// TwinCAT 3 PLC project SPS_1
// ProgramVersion: 3.1.4026.10
// CompilerDefines: VISU_USEPROPERTYINFO
// libraries:
//   Tc2_ModbusRTU, * (Beckhoff Automation GmbH)
//   Tc2_Standard, * (Beckhoff Automation GmbH)
//   Tc2_System, * (Beckhoff Automation GmbH)
//   Tc2_TcpIp, * (Beckhoff Automation GmbH)
//   Tc2_Utilities, * (Beckhoff Automation GmbH)
// project tree:
//   DUTs/01_Liste/01_Zustände/ eObjectAktorState.TcDUT, eSequenceState.TcDUT, eSkillState.TcDUT, eSystemState.TcDUT
//   DUTs/01_Liste/02_Commands/ eSkillCommand.TcDUT, eSystemCommand.TcDUT
//   DUTs/01_Liste/03_Konfiguration/ eRobMoveType.TcDUT, eRobPosType.TcDUT
//   DUTs/02_Schnittstellen/ I_State_Skill.TcIO, I_State_Object.TcIO
//   DUTs/03_Strukturen/01_Schnittstellen/ sKraftVariablen.TcDUT, sRoboterProzessVariablen.TcDUT, sSmartGreiferProzessVariablen.TcDUT
//   DUTs/03_Strukturen/02_Objektintern/01_FB_Roboter/ sPositionArrays.TcDUT, sPositionValues.TcDUT, sRealTimeData.TcDUT
//   DUTs/03_Strukturen/02_Objektintern/02_FB_Kraftsensor/ Kraftvariablen.TcDUT (not stored), Request.TcDUT, Response_Parameters.TcDUT, Response_Values.TcDUT
//   DUTs/04_Union/ Array2_Int.TcDUT, Array8_LReal.TcDUT, Int_2Byte.TcDUT, String_Array256.TcDUT
//   / GlobalTextList.TcGTLO, PlcTask.TcTTO, Visualization Manager.TcVMO (not stored), VISU_TASK.TcTTO
//   GVLs/ GVL.TcGVL
//   POUs/01_Prozessmodell/01_Skills/01_Grundstruktur/ GrundstrukturSkill.TcPOU
//   POUs/01_Prozessmodell/01_Skills/02_Skills/00_Referenz/ Basis_Skill.TcPOU
//   POUs/01_Prozessmodell/01_Skills/02_Skills/01_Roboter/ Skill_Position_anfahren.TcPOU (not stored), Skill_Position_anfahren_erweitert.TcPOU
//   POUs/01_Prozessmodell/01_Skills/02_Skills/02_Greifer/ Skill_Greifer_Oeffnen.TcPOU, Skill_Greifer_Pos_Anfahren.TcPOU, Skill_Greifer_Schliessen.TcPOU
//   POUs/01_Prozessmodell/02_Sequenzen/ Seq_1.TcPOU, Seq_2.TcPOU
//   POUs/02_Anlagenmodell/01_Grundstruktur/ GrundstrukturObjekt.TcPOU
//   POUs/02_Anlagenmodell/02_Objektklassen/00_Referenz/ Basis_Objekt.TcPOU
//   POUs/02_Anlagenmodell/02_Objektklassen/ FB_Kraftsensor.TcPOU, FB_Roboter.TcPOU, FB_SmartGreifer.TcPOU
//   POUs/02_Anlagenmodell/ Anlage.TcPOU
//   POUs/03_Systemmodell/ Systemparameter.TcPOU, Zustandshandling.TcPOU
//   POUs/ MAIN.TcPOU
//   VISUs/00_Debug/ SystemState.TcVIS
// real-time tasks:
//   TASK PlcTask: cycle T#10ms, priority 20, ADS port 350
//   TASK VISU_TASK: cycle T#200000us, priority 30, ADS port 351
//   TASK PlcTask1: cycle T#10ms, priority 21, ADS port 352
//   TASK PlcTask2: cycle T#10ms, priority 22, ADS port 353
// I/O:
//   DEVICE Gerät 1 (EtherCAT), AmsNetId 147.87.172.51.2.1
//     Box 1 (BK1120)
// variable links:
//   SPS_3/SPS_3 Instance <-> Device 1 (EtherCAT)/Box 1 (BK1120)
//     PlcTask Inputs/Anlage.Gripper.Communication.InData/D[{0..21}] <-> Term 2 (KL6041)/Channel 1/Data In {0..21}  (22 links)
//     PlcTask Inputs/Anlage.Gripper.Communication.InData/Status <-> Term 2 (KL6041)/Channel 1/Status
//     PlcTask Outputs/Anlage.Gripper.Communication.OutData/Ctrl <-> Term 2 (KL6041)/Channel 1/Ctrl
//     PlcTask Outputs/Anlage.Gripper.Communication.OutData/D[{0..21}] <-> Term 2 (KL6041)/Channel 1/Data Out {0..21}  (22 links)

CONFIGURATION SPS_1
    RESOURCE PLC ON TwinCAT3
        TASK PlcTask(INTERVAL := T#10ms, PRIORITY := 20);
        TASK VISU_TASK(INTERVAL := T#200000us, PRIORITY := 30);
        PROGRAM MAIN WITH PlcTask : MAIN;
        PROGRAM VisuElems_Visu_Prg WITH VISU_TASK : VisuElems.Visu_Prg;
    END_RESOURCE
END_CONFIGURATION

// ---- DUTs/01_Liste/01_Zustände/eObjectAktorState.TcDUT
{attribute 'qualified_only'}
{attribute 'strict'}
{attribute 'to_string'}
TYPE eObjectAktorState :
(
	AUS 					:= 0,				// Das Objekt ist ausgeschalten
	BEREIT 					:= 1,				// Das Objekt ist eingeschalten und bereit
	MANUELL					:= 2,				// Das Objekt befindet sich im Manuell-Modus
	LAUFEND 				:= 3,				// Das Objekt ist aktiv
	ABGESCHLOSSEN_INTERN 	:= 4,				// Das Objekt hat den Prozess durchgeführt und hat selbständig gestoppt
	ABGESCHLOSSEN_EXTERN	:= 5,				// Das Objekt wurde durch den Skill gestoppt (ERREICHT / LIMIT)
	GESTOPPT 				:= 6,				// Das Objekt wurde durch das System gestoppt
	FEHLER					:= 7				// Es gibt einen Fehler bezüglich des Objektes
);
END_TYPE

// ---- DUTs/01_Liste/01_Zustände/eSequenceState.TcDUT
{attribute 'qualified_only'}
{attribute 'strict'}
{attribute 'to_string'}
TYPE eSequenceState  :
(
	BEREIT	 		:= 0,				// Der Skill ist bereit einen Prozess auszuführen (Startzustand)
	LAUFEND 		:= 1,				// Der Skill führt einen Prozess aus
	ABGESCHLOSSEN 	:= 2,				// Der Prozess wurde abgeschlossen (Durch Objekt abgeschlossen)
	FEHLER			:= 3				// Es gibt einen Fehler bezüglich des Prozesses 
);
END_TYPE

// ---- DUTs/01_Liste/01_Zustände/eSkillState.TcDUT
{attribute 'qualified_only'}
{attribute 'strict'}
{attribute 'to_string'}
TYPE eSkillState :
(
	BEREIT	 		:= 0,				// Der Skill ist bereit einen Prozess auszuführen (Startzustand)
	LAUFEND 		:= 1,				// Der Skill führt einen Prozess aus
	ABGESCHLOSSEN 	:= 2,				// Der Prozess wurde abgeschlossen (Durch Objekt abgeschlossen)
	FEHLER			:= 3,				// Es gibt einen Fehler bezüglich des Prozesses 
	LIMITE			:= 4,				// Grenzwert wurde überschritten und Prozess wurde abgebrochen
	ERREICHT		:= 5				// Prozessziel wurde erreicht und Prozess wurde durch Skill beendet  
);	
END_TYPE

// ---- DUTs/01_Liste/01_Zustände/eSystemState.TcDUT
{attribute 'qualified_only'}
{attribute 'strict'}
{attribute 'to_string'}
TYPE eSystemState :
(
	AUS 			:= 0,				// Das System ist ausgeschalten
	BEREIT 			:= 1,				// Das System ist eingeschalten und bereit einen Prozess durchzuführen
	LAUFEND 		:= 2,				// Ein Prozess wird ausgeführt
	GESTOPPT		:= 3,				// Ein Prozess wurde gestoppt
	FEHLER			:= 4				// Es gibt einen Fehler im System 
);
END_TYPE

// ---- DUTs/01_Liste/02_Commands/eSkillCommand.TcDUT
{attribute 'qualified_only'}
{attribute 'strict'}
{attribute 'to_string'}
TYPE eSkillCommand :
(
	KEINE		:= 0,
	STARTEN		:= 1,
	STOPPEN		:= 2,
	RESETTEN 	:= 3
);
END_TYPE

// ---- DUTs/01_Liste/02_Commands/eSystemCommand.TcDUT
{attribute 'qualified_only'}
{attribute 'strict'}
{attribute 'to_string'}
TYPE eSystemCommand :
(
	KEINE		:= 0,
	AUSCHALTEN 	:= 1,
	EINSCHALTEN := 2,
	STOPPEN		:= 3,
	RESETTEN	:= 4
);
END_TYPE

// ---- DUTs/01_Liste/03_Konfiguration/eRobMoveType.TcDUT
{attribute 'qualified_only'}
{attribute 'strict'}
{attribute 'to_string'}
TYPE eRobMoveType :
(
	LinearToolSpace 			:= 0,		// Move to position (linear in tool-space)
	LinearJointSpace 			:= 1,		// Move to position (linear in joint-space)
	CircularToolSpace 			:= 2,		// Move Circular: Move to position (circular in tool-space)
	BlendCircularMoveLinear		:= 3		// Move Process
);
END_TYPE

// ---- DUTs/01_Liste/03_Konfiguration/eRobPosType.TcDUT
{attribute 'qualified_only'}
{attribute 'strict'}
{attribute 'to_string'}
TYPE eRobPosType :
(
	Absolut := 0,			// Absolute Bewegung bezogen auf Basis-Koordinatensystem
	Relativ := 1			// Relative Bewegung bezogen auf aktuelle Position
);
END_TYPE

// ---- DUTs/03_Strukturen/01_Schnittstellen/sKraftVariablen.TcDUT
TYPE sKraftVariablen :
STRUCT
	Fx					:LREAL;							// Kraft in X-Richtung 
	Fy					:LREAL;							// Kraft in Y-Richtung 
	Fz					:LREAL;							// Kraft in Z-Richtung 
END_STRUCT
END_TYPE

// ---- DUTs/03_Strukturen/01_Schnittstellen/sRoboterProzessVariablen.TcDUT
TYPE sRoboterProzessVariablen :
STRUCT
	q1					:LREAL;				// X-Koordinate oder Gelenkwinkel 1
	q2					:LREAL;				// Y-Koordinate oder Gelenkwinkel 2
	q3					:LREAL;				// Z-Koordinate oder Gelenkwinkel 3
	q4					:LREAL;				// Orintierung um X-Achse oder Gelenkwinkel 4
	q5					:LREAL;				// Orientierung um Y-Achse oder Gelenkwinkel 5
	q6					:LREAL;				// Orientierung um Z-Achse oder Gelenkwinkel 6
	v					:LREAL;				// Geschwindigkeit
	a					:LREAL;				// Beschleunigung
	PosTyp				:eRobPosType;		// Position-Typ definieren (Absolut / Relativ)		
	MoveTyp				:eRobMoveType;		// Bewegungsart definieren (Linear / Circular etc.)
END_STRUCT
END_TYPE

// ---- DUTs/03_Strukturen/01_Schnittstellen/sSmartGreiferProzessVariablen.TcDUT
TYPE sSmartGreiferProzessVariablen :
STRUCT
	Pos				:USINT;			// Position von Greifer in mm
	Geschw			:USINT;			// Geschwindigkeit in %
	F				:USINT;			// Kraft in %
END_STRUCT
	
END_TYPE

// ---- DUTs/03_Strukturen/02_Objektintern/01_FB_Roboter/sPositionArrays.TcDUT
TYPE sPositionArrays :
STRUCT
	q1		: ARRAY[0..7] OF BYTE;
	q2		: ARRAY[0..7] OF BYTE;
	q3		: ARRAY[0..7] OF BYTE;
	q4		: ARRAY[0..7] OF BYTE;
	q5		: ARRAY[0..7] OF BYTE;
	q6		: ARRAY[0..7] OF BYTE;
END_STRUCT
END_TYPE

// ---- DUTs/03_Strukturen/02_Objektintern/01_FB_Roboter/sPositionValues.TcDUT
TYPE sPositionValues :
STRUCT
	q1			:LREAL;
	q2			:LREAL;
	q3			:LREAL;
	q4			:LREAL;
	q5			:LREAL;
	q6			:LREAL;
END_STRUCT
END_TYPE

// ---- DUTs/03_Strukturen/02_Objektintern/01_FB_Roboter/sRealTimeData.TcDUT
TYPE sRealTimeData :
STRUCT
	messageSize 				: ARRAY[0..3] OF BYTE;
	
	timestamp 					: ARRAY[0..7] OF BYTE;
	
	//qTarget 					: ARRAY[0..47] OF BYTE;
	qTargetQ1 					: ARRAY[0..7] OF BYTE;
	qTargetQ2 					: ARRAY[0..7] OF BYTE;
	qTargetQ3 					: ARRAY[0..7] OF BYTE;
	qTargetQ4 					: ARRAY[0..7] OF BYTE;
	qTargetQ5 					: ARRAY[0..7] OF BYTE;
	qTargetQ6 					: ARRAY[0..7] OF BYTE;
	
	qdTarget 					: ARRAY[0..47] OF BYTE;
	
	qddTarget 					: ARRAY[0..47] OF BYTE;
	
	iTarget 					: ARRAY[0..47] OF BYTE;
	
	mTarget 					: ARRAY[0..47] OF BYTE;
	
	//qActual 					: ARRAY[0..47] OF BYTE;
	qActualQ1 					: ARRAY[0..7] OF BYTE;
	qActualQ2 					: ARRAY[0..7] OF BYTE;
	qActualQ3 					: ARRAY[0..7] OF BYTE;
	qActualQ4 					: ARRAY[0..7] OF BYTE;
	qActualQ5 					: ARRAY[0..7] OF BYTE;
	qActualQ6 					: ARRAY[0..7] OF BYTE;
	
	//qdActual 					: ARRAY[0..47] OF BYTE;
	qdActualQ1 					: ARRAY[0..7] OF BYTE;
	qdActualQ2 					: ARRAY[0..7] OF BYTE;
	qdActualQ3 					: ARRAY[0..7] OF BYTE;
	qdActualQ4 					: ARRAY[0..7] OF BYTE;
	qdActualQ5 					: ARRAY[0..7] OF BYTE;
	qdActualQ6 					: ARRAY[0..7] OF BYTE;
	
	iActual 					: ARRAY[0..47] OF BYTE;
	
	toolAccelerometerValues 	: ARRAY[0..23] OF BYTE;
	
	unused_1					: ARRAY[0..119] OF BYTE;
	
	tcpForce 					: ARRAY[0..47] OF BYTE;
	
	//toolVector 					: ARRAY[0..47] OF BYTE;
	toolVectorQ1 				: ARRAY[0..7] OF BYTE;
	toolVectorQ2 				: ARRAY[0..7] OF BYTE;
	toolVectorQ3 				: ARRAY[0..7] OF BYTE;
	toolVectorQ4 				: ARRAY[0..7] OF BYTE;
	toolVectorQ5 				: ARRAY[0..7] OF BYTE;
	toolVectorQ6 				: ARRAY[0..7] OF BYTE;
	
	tcpSpeed 					: ARRAY[0..47] OF BYTE;
	
	digitalInputBits 			: ARRAY[0..7] OF BYTE;
	
	unused_2					: ARRAY[0..119] OF BYTE;
END_STRUCT
END_TYPE

// ---- DUTs/03_Strukturen/02_Objektintern/02_FB_Kraftsensor/Request.TcDUT
TYPE Request :
STRUCT
	Command			:UINT;		// Value according to the command table
	Data			:ARRAY[0..18] OF UINT := [0];		
END_STRUCT
END_TYPE

// ---- DUTs/03_Strukturen/02_Objektintern/02_FB_Kraftsensor/Response_Parameters.TcDUT
TYPE Response_Parameters :
STRUCT
	Header				:UINT;			// Fixed 0x1234
	Unit_Force			:USINT;			// The unit of the calculated Force values
	Unit_Torque			:USINT;			// The unit of the calculated Torque values
	CPF					:UDINT;			// Counts per Force value
	CPT					:UDINT;			// Counts per Torque value
	ScaleFactorFx		:UINT;			// Additional scaling factor (for the Fx,Fy,Fz,Tx,Ty,Tz)
	ScaleFactorFy		:UINT;			// Additional scaling factor (for the Fx,Fy,Fz,Tx,Ty,Tz)
	ScaleFactorFz		:UINT;			// Additional scaling factor (for the Fx,Fy,Fz,Tx,Ty,Tz)
	ScaleFactorTx		:UINT;			// Additional scaling factor (for the Fx,Fy,Fz,Tx,Ty,Tz)
	ScaleFactorTy		:UINT;			// Additional scaling factor (for the Fx,Fy,Fz,Tx,Ty,Tz)
	ScaleFactorTz		:UINT;			// Additional scaling factor (for the Fx,Fy,Fz,Tx,Ty,Tz)
END_STRUCT
END_TYPE

// ---- DUTs/03_Strukturen/02_Objektintern/02_FB_Kraftsensor/Response_Values.TcDUT
TYPE Response_Values :
STRUCT
	Header				:UINT;			// Fixed 0x1234
	Status				:UINT;			// Status word of the sensor and Compute Box
	Fx					:INT;			// X-axis force in 32 bit Counts*
	Fy					:INT;			// Y-axis force in 32 bit Counts*
	Fz					:INT;			// Z-axis force in 32 bit Counts*
	Tx					:INT;			// X-axis torque in 32 bit Counts* (0 if not available)
	Ty					:INT;			// Y-axis torque in 32 bit Counts* (0 if not available)
	Tz					:INT;			// Z-axis torque in 32 bit Counts* (0 if not available)
END_STRUCT
END_TYPE

// ---- DUTs/04_Union/Array2_Int.TcDUT
TYPE Array2_Int :
UNION
	arrByte 		:ARRAY[0..1] OF BYTE;
	sValue			:INT; 
END_UNION
END_TYPE

// ---- DUTs/04_Union/Array8_LReal.TcDUT
TYPE Array8_LReal :
UNION
	arrByte			:ARRAY[0..7] OF BYTE;
	rValue			:LREAL;
END_UNION
END_TYPE

// ---- DUTs/04_Union/Int_2Byte.TcDUT
TYPE Int_2Byte :
UNION
	sValue			:INT; 
	arrByte 		:ARRAY[0..1] OF BYTE;
END_UNION
END_TYPE

// ---- DUTs/04_Union/String_Array256.TcDUT
TYPE String_Array256 :
UNION
	sValue			:STRING; 
	arrByte 		:ARRAY[0..255] OF BYTE;
END_UNION
END_TYPE

// ---- GVLs/GVL.TcGVL
{attribute 'qualified_only'}
VAR_GLOBAL
	// Schnittstellenvariablen 
		// System: 
		SystemState								:eSystemState; 
		SystemCommand							:eSystemCommand; 
		Error									:BOOL;
		
		// Kontrollvariablen: 
		Reset									:BOOL;
		
		// Prozessvariablen
		eKraftLimitValue						:sKraftVariablen;
		eKraftErreichtValue						:sKraftVariablen;
		
		
		// SkillStates
		
		// ObjectStates
		Robot_State								:eObjectAktorState;
		Greifer_State							:eObjectAktorState;
		Sensor_State							:eObjectAktorState;
		
			
		
		
		
END_VAR

// ---- DUTs/02_Schnittstellen/I_State_Skill.TcIO
INTERFACE I_State_Skill

PROPERTY P_State : eSkillState
GET
END_GET
END_PROPERTY

END_INTERFACE

// ---- DUTs/02_Schnittstellen/I_State_Object.TcIO
INTERFACE I_State_Object

PROPERTY P_State : eObjectAktorState
GET
END_GET
END_PROPERTY

END_INTERFACE

// ---- POUs/MAIN.TcPOU
PROGRAM MAIN
VAR
	TestAblauf				:Seq_2;
	
	Execute					:BOOL;		
	Position_1				:sRoboterProzessVariablen;
	Position_2				:sRoboterProzessVariablen;
	Position_3				:sRoboterProzessVariablen;

	
	TestSystem				:eSystemCommand; 
	TestSkill				:eSkillCommand; 
	TestVariablen			:sSmartGreiferProzessVariablen;
	
	Param1					:sSmartGreiferProzessVariablen;
	Param2					:sSmartGreiferProzessVariablen;
	Param3					:sSmartGreiferProzessVariablen;
	Param4					:sSmartGreiferProzessVariablen;
		
END_VAR

Zustandshandling();
Anlage();
Systemparameter();


Position_1.q1 := -0.3;
Position_1.q2 := 0.5;
Position_1.q3 := 0.42;
Position_1.q4 := 120;
Position_1.q5 := -132;
Position_1.q6 := 0;
Position_1.a := 0.05;
Position_1.v := 0.05;
Position_1.MoveTyp := 3;
Position_1.PosTyp := 0;

Position_2.q1 := 0.4;
Position_2.q2 := 0.52;
Position_2.q3 := 0.42;
Position_2.q4 := 120;
Position_2.q5 := -132;
Position_2.q6 := 0;
Position_2.a := 0.05;
Position_2.v := 0.05;
Position_2.MoveTyp := 3;
Position_2.PosTyp := 0;

Position_3.q1 := 0.05;
Position_3.q2 := 0.68;
Position_3.q3 := 0.42;
Position_3.q4 := 120;
Position_3.q5 := -132;
Position_3.q6 := 0;
Position_3.a := 0.05;
Position_3.v := 0.05;
Position_3.MoveTyp := 3;
Position_3.PosTyp := 0;

GVL.eKraftLimitValue.Fz := -40;

TestAblauf(
	bExecute := Execute,
	iSysCommand := GVL.SystemCommand,
	Position_1 := Position_1,
	Position_2 := Position_2,
	Position_3 := Position_3);

END_PROGRAM

// ---- POUs/01_Prozessmodell/02_Sequenzen/Seq_2.TcPOU
FUNCTION_BLOCK Seq_2
VAR_INPUT
	// Basis-Inputs
	bExecute			:BOOL;				// Trigger für Ausführung von Sequenz
	iSysCommand			:eSystemCommand;	// Steuerungsvariabel von System (Resetten)
	
	// Prozess-Inputs 
	Position_1			:sRoboterProzessVariablen;
	Position_2			:sRoboterProzessVariablen;
	Position_3			:sRoboterProzessVariablen;
	
END_VAR
VAR_OUTPUT
	bDone				:BOOL;				// Information ob Sequenz ausgfeührt wurde
	bBusy				:BOOL;				// Information ob Sequenz im Moment ausgeführt wird
	bError				:BOOL;				// Information ob sich Sequenz in Fehlerzustand befindet
END_VAR
VAR
	// Sequenz-Zustände
	iState				:eSequenceState;
	
	// Startvariablen (FB soll nur bei einer steigenden Flanke gestartet werden)
	fTrigger			:R_TRIG;			// Erkennung einer steigenden Flanke für den Starte
	fSwitch				:SR;				// Setzen des Signals
	bSwitchResett		:BOOL;				// Resetten des Signals
	
	// Zustandsvariablen
	bStarten			:BOOL;
	bStoppen			:BOOL;
	bResetten			:BOOL;
	
	// Management-Variablen:
	bFinished			:BOOL;
	bInit				:BOOL;
	
	// Skill-Instanziierungen
	P2P_Movement		:Skill_Position_anfahren_erweitert;
	Position			:sRoboterProzessVariablen;
END_VAR

// Aufrufen von Skills und Ablauf
Ablauf();	
Skills();

//_______________________________________________________________
// Reaktion auf Fehler
IF bError THEN
	iState := 3;
END_IF	

// Reaktion auf Input-Variablen: 
	// Starten
	fTrigger(CLK := bExecute);
	fSwitch(Set1 := fTrigger.Q);
	
	IF fSwitch.Q1 THEN
		bStarten := TRUE;
	ELSE
		bStarten := FALSE;
	END_IF
	
	// Stoppen
	IF iSysCommand = 3 THEN
		bStoppen := TRUE;	
	ELSE 
		bStoppen := FALSE;	
	END_IF
	
	// Stoppen
	IF iSysCommand = 4 THEN
		bResetten := TRUE;	
	ELSE 
		bResetten := FALSE;	
	END_IF



//_______________________________________________________________
// Zustandsmanagement
CASE iState OF 
	0:	// BEREIT
			// DO	
			fSwitch.RESET := FALSE;
				
			// TRANSITION
			IF bStarten THEN
				fSwitch.RESET := TRUE;
				iState := 1;																							// Starten des Objektes 
			END_IF
	// ________________________________________________________________________________			
	1:	// LAUFEND
			// DO
			bBusy := TRUE;	

			IF bStoppen THEN
				SFCReset := TRUE;
				bBusy := FALSE;
			END_IF	
			
			// TRANSITION
			IF bFinished THEN
				bFinished := FALSE;
				bBusy := FALSE;
				iState := 2;
			END_IF
			
			IF bInit THEN
				bInit := FALSE;
				SFCReset := FALSE;
				iState := 0;
			END_IF

	// ________________________________________________________________________________					
	2:	// ABGESCHLOSSEN
			// DO
			bDone := TRUE;			
						
			// TRANSITION
			IF bDone THEN
				bDone := FALSE;
				iState := 0;
			END_IF
	// ________________________________________________________________________________					
	3:	// FEHLER
			// DO
			bDone := FALSE;
			bBusy := FALSE;
			
			// TRANSITION
			IF bResetten THEN
				bError := FALSE;
				iState := 0;
			END_IF
			
END_CASE

ACTION Ablauf:
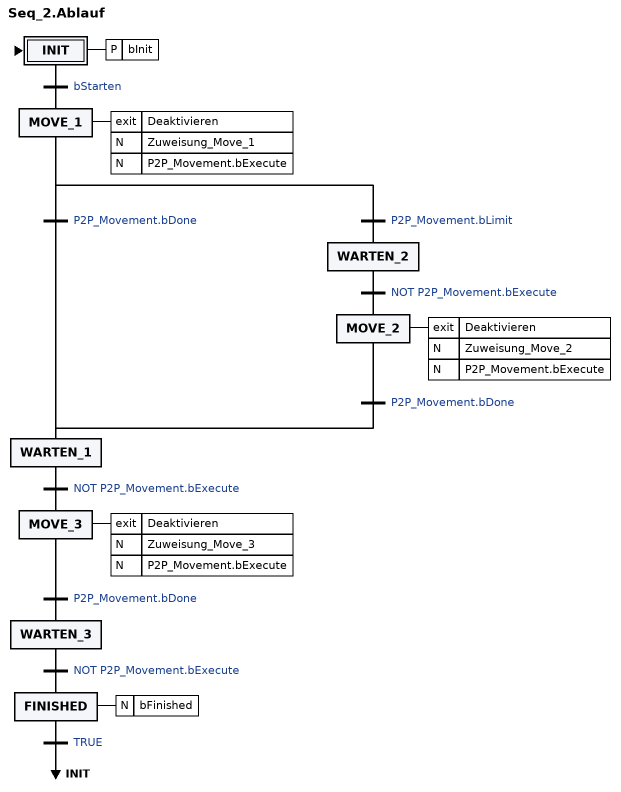
INITIAL_STEP INIT:
    bInit(P);
END_STEP
TRANSITION FROM INIT TO MOVE_1
    := bStarten;
END_TRANSITION
STEP MOVE_1:
    Deaktivieren(P0);  // exit action
    Zuweisung_Move_1(N);
    P2P_Movement.bExecute(N);
END_STEP
TRANSITION FROM MOVE_1 TO WARTEN_1
    := P2P_Movement.bDone;
END_TRANSITION
TRANSITION FROM MOVE_1 TO WARTEN_2
    := P2P_Movement.bLimit;
END_TRANSITION
STEP WARTEN_2:
END_STEP
TRANSITION FROM WARTEN_2 TO MOVE_2
    := NOT P2P_Movement.bExecute;
END_TRANSITION
STEP MOVE_2:
    Deaktivieren(P0);  // exit action
    Zuweisung_Move_2(N);
    P2P_Movement.bExecute(N);
END_STEP
TRANSITION FROM MOVE_2 TO WARTEN_1
    := P2P_Movement.bDone;
END_TRANSITION
STEP WARTEN_1:
END_STEP
TRANSITION FROM WARTEN_1 TO MOVE_3
    := NOT P2P_Movement.bExecute;
END_TRANSITION
STEP MOVE_3:
    Deaktivieren(P0);  // exit action
    Zuweisung_Move_3(N);
    P2P_Movement.bExecute(N);
END_STEP
TRANSITION FROM MOVE_3 TO WARTEN_3
    := P2P_Movement.bDone;
END_TRANSITION
STEP WARTEN_3:
END_STEP
TRANSITION FROM WARTEN_3 TO FINISHED
    := NOT P2P_Movement.bExecute;
END_TRANSITION
STEP FINISHED:
    bFinished(N);
END_STEP
TRANSITION FROM FINISHED TO INIT
    := TRUE;
END_TRANSITION
// branch label Branch0_Ablauf
END_ACTION

ACTION Deaktivieren:
P2P_Movement.bExecute := FALSE;
END_ACTION

ACTION Skills:
P2P_Movement(
    iSysCommand := GVL.SystemCommand,
    iObjState := Anlage.UR5.P_State,
    iSysState := GVL.SystemState,
    sProzessvariablen := Position,
    bLimitTrig := Anlage.HEX_E.P_Limit,
    bErreichtTrig := Anlage.HEX_E.P_Erreicht); // Skill_Position_anfahren_erweitert
Anlage.UR5.iSkillCommand_1 := P2P_Movement.iSkillCommand;
Anlage.UR5.Prozessvariablen := P2P_Movement.sObjektvariablen;
END_ACTION

ACTION Zuweisung_Move_1:
Position := Position_1;
END_ACTION

ACTION Zuweisung_Move_2:
Position := Position_2;
END_ACTION

ACTION Zuweisung_Move_3:
Position := Position_3;
END_ACTION

END_FUNCTION_BLOCK

// ---- POUs/01_Prozessmodell/01_Skills/02_Skills/01_Roboter/Skill_Position_anfahren_erweitert.TcPOU
FUNCTION_BLOCK Skill_Position_anfahren_erweitert EXTENDS GrundstrukturSkill
VAR_INPUT 
	sProzessvariablen			:sRoboterProzessVariablen;
	bLimitTrig					:BOOL;
	bErreichtTrig				:BOOL;
END_VAR
VAR_OUTPUT
	sObjektvariablen			:sRoboterProzessVariablen;
END_VAR
VAR
	
END_VAR

// Fehlerüberwachung
IF bFehler THEN
	iState := 3;
END_IF

//_______________________________________________________________
// Reaktion auf Input-Variablen:
	// Starten
	fTrigger(CLK := bExecute);
	fSwitch(Set1 := fTrigger.Q);
	
	IF fSwitch.Q1 AND iSysState = 1 THEN
		bStarten := TRUE;
		fSwitch.RESET := TRUE;
	ELSE
		bStarten := FALSE;
		fSwitch.RESET := FALSE;
	END_IF

	// Stoppen
	IF iSysCommand = 3 THEN
		bStoppen := TRUE;
	ELSE 
		bStoppen := FALSE;
	END_IF

	// Resetten 
	IF iSysCommand = 4 THEN
		bResetten := TRUE;
	ELSE
		bResetten := FALSE;
	END_IF
	
	// Limit 
	IF bLimitTrig THEN
		bLimitReached := TRUE;
	ELSE
		bLimitReached := FALSE;
	END_IF
	// Erreicht
	IF bErreichtTrig THEN
		bTargetReached := TRUE;
	ELSE 
		bTargetReached := FALSE;
	END_IF
	

//_______________________________________________________________
// Zustandsmanagement
CASE iState OF 
0: 	// BEREIT
		// DO
		bDone := FALSE;	
	
		IF bStarten THEN
			IF ParameterError OR PositionError THEN
				bError := TRUE;
			ELSE	
				sObjektvariablen := sProzessvariablen;
				iSkillCommand := 1;																						// Starten des Objektes 
			END_IF		
		END_IF	
		
		IF iObjState = 3 THEN																					// Resetten von Startsignal
			bGestartet := TRUE;
		END_IF
			
		// TRANSITION	
		IF bGestartet THEN
			bGestartet := FALSE;
			iState := 1;																								// Objekt wurde gestartet
		END_IF
// _________________________________________________________________________________________________________________________
1: 	// LAUFEND
		// DO
		iSkillCommand := 0;
		bBusy := TRUE;																									// Skill wird ausgeführt
		
		
		IF bTargetReached OR bLimitReached THEN																			// Prüfen ob Prozessziel erreicht wurde
			iSkillCommand := 2;
		END_IF
		
		IF iObjState = 4 THEN																							// Objekt hat Prozess abgeschlossen
			bBusy := FALSE;																									// Skill wird nicht mehr ausgeführt			
			bObjektFertig := TRUE;																							// Objekt ist fertig und wieder bereit
		END_IF
		
		IF bStoppen THEN																							// Transition wenn System das Orbjekt stoppt
			bBusy := FALSE;																									// Skill wird nicht mehr ausgeführt
		END_IF
		
		IF bLimitReached AND iObjState = 5 THEN																			// Objekt wurde duch Skill gestoppt - LIMIT
			iSkillCommand := 0;																								// Zurücksetzen von Command																						// Zurücksetzen von Information	
			bBusy := FALSE;																									// Skill wird nicht mehr ausgeführt
			bLimitErreicht := TRUE;	
		END_IF
		
		IF bTargetReached AND iObjState = 5 THEN																			// Objekt wurde duch Skill gestoppt - LIMIT
			iSkillCommand := 0;																									// Zurücksetzen von Command
			bTargetReached := FALSE;																							// Zurücksetzen von Information	
			bBusy := FALSE;																										// Skill wird nicht mehr ausgeführt
			bWertErreicht := TRUE;	
		END_IF
			
		// TRANSITION 
		IF bObjektFertig THEN																							// Transition zu ABGESCHLOSSEN
			bObjektFertig := FALSE;																							// Skill wird nicht mehr ausgeführt
			iState := 2;																									// Objekt ist fertig und wieder bereit
		END_IF
		
		IF bGestoppt THEN																									// Transition zu BEREIT
			bGestoppt := FALSE;																							
			iState := 0;
		END_IF
		
		IF bLimitErreicht THEN																							// Transition zu LIMIT
			bLimitErreicht := FALSE;
			iState := 4;
		END_IF
		
		IF bWertErreicht THEN																							// Transition zu ERREICHT																						// Skill wird nicht mehr ausgeführt
			bWertErreicht := FALSE;
			iState := 5;
		END_IF
			
// _________________________________________________________________________________________________________________________			
2: 	// ABGESCHLOSSEN
		// DO																												// Skill wurde erfolgreich ausgeführt
		iSkillCommand := 3;
		bDone := TRUE;																										// Objekt resetten
		
		IF iObjState = 1 THEN
			iSkillCommand := 0;																								// Zurücksetzen von Command
			bSkillFertig := TRUE;											
		END_IF
			
		//  TRANSITION
		IF bSkillFertig THEN
			bSkillFertig := FALSE;																							// Zurücksetzen von Skill																																										// Resetten von Objekt
			iState := 0;
		END_IF
		
// _________________________________________________________________________________________________________________________
3: 	// FEHLER
		// DO 
		iSkillCommand := 0;	
		bDone := FALSE;
		bBusy := FALSE;
		
		IF ParameterError THEN
			// Setzen von ErrorID
		END_IF
		
		IF PositionError THEN
			// Setzen von ErrorID
		END_IF
		
		// TRANSITION
		IF bResetten THEN
			iState := 0;
		END_IF
		
// _________________________________________________________________________________________________________________________			
4: 	// LIMIT
		// DO 
		bLimit := TRUE;																									// Limit wurde erreicht
		iSkillCommand := 3;																								// Objekt resetten
		
		IF iObjState = 1 THEN																							// Objekt wurde geresettet
			iSkillCommand := 0;																								// Zurücksetzen von Command
			bDone := FALSE;																									// Zurücksetzen von Skill
			bResetten := TRUE;								
		END_IF
	
		// TRANSITION
		IF bResetten THEN
			bResetten := FALSE;
			bLimit := FALSE;																							// Zurücksetzen von Output-Variable
			iState := 0;
		END_IF
		
// _________________________________________________________________________________________________________________________
5: 	// ERREICHT		
		// DO 
		bDone := TRUE;																								// Skill wurde erfolgreich ausgeführt
		
		iSkillCommand := 3;																								// Objekt resetten
		
		IF iObjState = 1 THEN																							// Objekt wurde geresettet
			iSkillCommand := 0;																								// Zurücksetzen von Command
			bDone := FALSE;																									// Zurücksetzen von Skill
			bSkillFertig := TRUE;									
		END_IF
		
		// TRANSITION
		IF bSkillFertig THEN
			bSkillFertig := FALSE;
			iState := 0;
		END_IF

END_CASE

TRANSITION ParameterError:
IF sProzessvariablen.a = 0 OR sProzessvariablen.v = 0 THEN
	ParameterError := TRUE;
END_IF
END_TRANSITION

TRANSITION PositionError:
IF sProzessvariablen.q1 = 0 AND sProzessvariablen.q2 = 0 AND sProzessvariablen.q3 = 0 AND sProzessvariablen.q4 = 0 AND sProzessvariablen.q5 = 0 AND sProzessvariablen.q6 = 0 THEN
	PositionError := TRUE;
END_IF
END_TRANSITION

END_FUNCTION_BLOCK

// ---- POUs/01_Prozessmodell/01_Skills/01_Grundstruktur/GrundstrukturSkill.TcPOU
FUNCTION_BLOCK GrundstrukturSkill IMPLEMENTS I_State_Skill
VAR_INPUT
	bExecute			:BOOL;				// Trigger für Ausführung von Skill
	iSysCommand			:eSystemCommand;	// Steuerungsvariabel von System (Resetten)
	iObjState			:eObjectAktorState;		// Information über Zustand von Objekt
	iSysState			:eSystemState;		// Information über Zustand von System
END_VAR
VAR_OUTPUT
	iSkillCommand		:eSkillCommand;		// Steuerungsvariable für Anlagenmodell
	bDone				:BOOL;				// Information ob Skill ausgfeührt wurde
	bBusy				:BOOL;				// Information ob Skill im Moment ausgeführt wird
	bLimit				:BOOL;				// Information ob Skill an einem Limit angekommen ist
	bError				:BOOL;				// Information ob sich Skill in Fehlerzustand befindet
	iErrorID			:INT;				// Information um welchen Fehler es sich handelt
END_VAR
VAR
	// Managementvariablen
	iState				:eSkillState;		// Information über Zustand von Skill
	bTargetReached		:BOOL;				// Information ob Prozessziel erreicht wurde
	bLimitReached		:BOOL;				// Information ob Limit erreicht wurde
	
	// Startvariablen (FB soll nur bei einer steigenden Flanke gestartet werden)
	fTrigger			:R_TRIG;			// Erkennung einer steigenden Flanke für den Starte
	fSwitch				:SR;				// Setzen des Signals
	
	// Managementvariablen 
	bGestartet			:BOOL;
	bGestoppt			:BOOL;
	
	// Zustandsvariablen
	bStarten			:BOOL;
	bStoppen			:BOOL;
	bObjektFertig		:BOOL;
	bWertErreicht		:BOOL;				
	bLimitErreicht		:BOOL;				
	bSkillFertig		:BOOL;
	bFehler				:BOOL;
	bResetten			:BOOL;
	
	
END_VAR

PROPERTY P_State : eSkillState
GET
P_State := iState;
END_GET
END_PROPERTY

END_FUNCTION_BLOCK

// ---- POUs/02_Anlagenmodell/Anlage.TcPOU
PROGRAM Anlage
VAR_INPUT
	UR5				:FB_Roboter;
	Gripper			:FB_SmartGreifer;
	HEX_E			:FB_Kraftsensor; 
END_VAR

VAR
END_VAR

UR5(
    iSysCommand := GVL.SystemCommand,
    iSysState := GVL.SystemState,
    sIP := '192.168.1.100',
    iPort_Prim := 30002,
    iPort_RT := 30003); // FB_Roboter
Gripper(iSysState := GVL.SystemState, iSysCommand := GVL.SystemCommand); // FB_SmartGreifer
HEX_E(iSysState := GVL.SystemState, iSysCommand := GVL.SystemCommand, sIP := '192.168.1.1', iPort := 49151); // FB_Kraftsensor

END_PROGRAM

// ---- POUs/02_Anlagenmodell/02_Objektklassen/FB_Roboter.TcPOU
FUNCTION_BLOCK FB_Roboter EXTENDS GrundstrukturObjekt
VAR_INPUT
	// Kommunikationsvariablen
	sIP						:T_IPv4Addr;
	iPort_Prim				:UINT;
	iPort_RT				:UINT;
	
	// Prozessvariablen
	Prozessvariablen		:sRoboterProzessVariablen;
END_VAR

VAR_OUTPUT
END_VAR

VAR
	// Instanziierung von Kommunikationsbausteine
	Connect					:FB_SocketConnect;
	Disconnect				:FB_SocketCloseALL;
	Send_START				:FB_SocketSend;
	Send_STOP				:FB_SocketSend;
	Connect_RT				:FB_SocketConnect;
	Receive_RT				:FB_SocketReceive;
	Disconnect_RT			:FB_SocketClose;
	
	// Kommunikationsvariablen
	sSrvNetId   			:T_AmsNetId := '';
	tTimeout    			:TIME := T#45S;(*!!!*)
	hSocket    				:T_HSOCKET;
	hSocket_RT    			:T_HSOCKET;
	
	// Managementvariablen
	bEingeschalten 			:BOOL;
	bAusgeschalten			:BOOL;
	bAmStarten				:BOOL;
	bGestartet				:BOOL;
	bAmStoppen				:BOOL;
	bGestoppt				:BOOL;
	
	bTurnedOn 				:BOOL;
	
	bBewegungStoppen		:BOOL;
	
	Delay_1					:TON;
	Delay_2					:TON;
	
	bQ1						:BOOL;
	bQ2						:BOOL;
	bQ3						:BOOL;
	bQ4						:BOOL;
	bQ5						:BOOL;
	bQ6						:BOOL;
	
	bVQ1					:BOOL;
	bVQ2					:BOOL;
	bVQ3					:BOOL;
	bVQ4					:BOOL;
	bVQ5					:BOOL;
	bVQ6					:BOOL;
	
	// RealTimeDatenerfassung
	RT_State				:INT;							// RealTime-State-Variable
	ReceivedData			:sRealTimedata;					// Erhaltene Daten von Roboter
	nRecBytes				:UDINT;							// Anzahl der erhaltenen Bytes
	
	JointPositions			:sPositionValues;				// Ausgelesene aktuelle Joint-Positonen-Byte
	JointSpeed				:sPositionValues;				// Ausgelesene aktuelle Joint-Geschwindigkeit-Byte
	ToolPosition			:sPositionValues;				// Ausgelesene aktuelle Tool-Positonen-Byte
	
	TempJointPosRev			:sPositionArrays;				// Ausgelesene aktuelle Joint-Positonen-Byte (Reversed)
	TempJointVRev			:sPositionArrays;				// Ausgelesene aktuelle Joint-Geschwindigkeit-Byte (Reversed)	
	TempToolPosRev			:sPositionArrays;				// Ausgelesene aktuelle Tool-Positonen-Byte(Reversed)
	
	Joint					:Array8_LReal;					// Aktuelle Joint-Positonen
	JSpeed					:Array8_LReal;					// Aktuelle Joint-Geschwindgeit
	Tool					:Array8_LReal;					// Aktuelle Tool-Positionen
	m						:INT;							// Loop-Variable
	
	// Prozessdaten
	TargetPosition			:sPositionValues;				// Targetpositions
	bSetValues				:BOOL;							// Definiert ob Targetposition noch ermittelt werden muss
	
	test 					:BOOL;
END_VAR

// Instanziierungen
	Connect_RT(sSrvNetId := sSrvNetId,
							sRemoteHost := sIP,
							nRemotePort := iPort_RT,
							tTimeout := tTimeout,
							bError => bFehler,
							nErrId => iErrorID,
							hSocket => hSocket_RT);	
							
	Send_START(sSrvNetId := sSrvNetId,
			hSocket := hSocket,
			tTimeout := tTimeout,
			bError => bFehler,
			nErrId => iErrorID);
	Send_STOP(sSrvNetId := sSrvNetId,
			hSocket := hSocket,
			tTimeout := tTimeout,
			bError => bFehler,
			nErrId => iErrorID);
							
	Receive_RT(sSrvNetId := sSrvNetId,
							hSocket := hSocket_RT,
							cbLen := SIZEOF(ReceivedData),
							pDest := ADR(ReceivedData),
							tTimeout := tTimeout,
							bError => bFehler,
							nErrId => iErrorID,
							nRecBytes => nRecBytes);
							
	Disconnect_RT(sSrvNetId := sSrvNetId,
							hSocket := hSocket_RT,
							tTimeout := tTimeout,
							bError => bFehler,
							nErrId => iErrorID);

//____________________________________________________________________________________________
// Input-Command-Verwaltung
	// System
	IF iSysCommand = 2 AND iState = 0 THEN			// Objekt einschalten
		bEinschalten := TRUE;
	ELSE 
		bEinschalten := FALSE;
	END_IF
	
	IF iSysCommand = 1 AND iState = 1 THEN			// Objekt ausschalten
		bAusschalten := TRUE;		
	ELSE 
		bAusschalten := FALSE;		
	END_IF
	
	IF iSysCommand = 3 THEN							// Objekt beendet Prozess
		bStoppen := TRUE;
	ELSE
		bStoppen := FALSE;
	END_IF
	
	IF iSysCommand = 4 THEN							// System resettet Objekt
		bResettenSystem := TRUE;
	ELSE
		bResettenSystem := FALSE;
	END_IF
	
	// Skill
	IF iSkillCommand_1 = 1 THEN						// Skill startet Prozess
		bStarten := TRUE;
	ELSE 
		bStarten := FALSE;
	END_IF
	
	IF iSkillCommand_1 = 2 THEN						// Skill beendet Prozess
		bSkillFertig := TRUE;
	ELSE
		bSkillFertig := FALSE;
	END_IF
	
	IF iSkillCommand_1 = 3 THEN						// Skill resettet Objekt
 		bResettenSkill := TRUE;
	ELSE
		bResettenSkill := FALSE;
	END_IF




//____________________________________________________________________________________________
// Interner Methodenaufruf (Durch System oder Skill)
IF bEinschalten THEN
	bEingeschalten := Verbinden();
	bTurnedOn := TRUE;
ELSE 
	bEingeschalten := FALSE;
END_IF

IF bAusschalten THEN
	bAusgeschalten := Trennen();
	bTurnedOn := FALSE;
	RT_State := 0;
ELSE 
	bAusgeschalten := FALSE;
END_IF

//____________________________________________________________________________________________
// Datenerfassungsprozess
IF bTurnedOn THEN
	CASE RT_State OF 
		0:	// Connect to RealTimePort
				Connect_RT(bExecute := TRUE);			
					
				IF NOT Connect_RT.bBusy AND NOT Connect_RT.bError THEN
					Connect_RT.bExecute := FALSE;
					RT_State := 1;
				END_IF
		
		1:	// Get Data 
				Receive_RT(bExecute := TRUE);
			
				IF NOT Receive_RT.bBusy AND NOT Receive_RT.bError THEN
					Receive_RT.bExecute := FALSE;
					RT_State := 2;
				END_IF
				
		2:	// Use Data
				m := 0;
		
				// Reverse Array
				FOR m := 0 TO 7 DO
					TempJointPosRev.q1[m] := ReceivedData.qActualQ1[7 - m];
					TempJointPosRev.q2[m] := ReceivedData.qActualQ2[7 - m];
					TempJointPosRev.q3[m] := ReceivedData.qActualQ3[7 - m];
					TempJointPosRev.q4[m] := ReceivedData.qActualQ4[7 - m];
					TempJointPosRev.q5[m] := ReceivedData.qActualQ5[7 - m];
					TempJointPosRev.q6[m] := ReceivedData.qActualQ6[7 - m];
					
					TempJointVRev.q1[m] := ReceivedData.qdActualQ1[7 - m];
					TempJointVRev.q2[m] := ReceivedData.qdActualQ2[7 - m];
					TempJointVRev.q3[m] := ReceivedData.qdActualQ3[7 - m];
					TempJointVRev.q4[m] := ReceivedData.qdActualQ4[7 - m];
					TempJointVRev.q5[m] := ReceivedData.qdActualQ5[7 - m];
					TempJointVRev.q6[m] := ReceivedData.qdActualQ6[7 - m];
					
					TempToolPosRev.q1[m] := ReceivedData.toolVectorQ1[7 - m];
					TempToolPosRev.q2[m] := ReceivedData.toolVectorQ2[7 - m];
					TempToolPosRev.q3[m] := ReceivedData.toolVectorQ3[7 - m];
					TempToolPosRev.q4[m] := ReceivedData.toolVectorQ4[7 - m];
					TempToolPosRev.q5[m] := ReceivedData.toolVectorQ5[7 - m];
					TempToolPosRev.q6[m] := ReceivedData.toolVectorQ6[7 - m];
				END_FOR
			
				Joint.arrByte := TempJointPosRev.q1;
				JointPositions.q1 := RAD_TO_DEG(Joint.rValue);
				Joint.arrByte := TempJointPosRev.q2;
				JointPositions.q2 := RAD_TO_DEG(Joint.rValue);
				Joint.arrByte := TempJointPosRev.q3;
				JointPositions.q3 := RAD_TO_DEG(Joint.rValue);
				Joint.arrByte := TempJointPosRev.q4;
				JointPositions.q4 := RAD_TO_DEG(Joint.rValue);
				Joint.arrByte := TempJointPosRev.q5;
				JointPositions.q5 := RAD_TO_DEG(Joint.rValue);
				Joint.arrByte := TempJointPosRev.q6;
				JointPositions.q6 := RAD_TO_DEG(Joint.rValue);
				
				JSpeed.arrByte := TempJointVRev.q1;
				JointSpeed.q1 := JSpeed.rValue;
				JSpeed.arrByte := TempJointVRev.q2;
				JointSpeed.q2 := JSpeed.rValue;
				JSpeed.arrByte := TempJointVRev.q3;
				JointSpeed.q3 := JSpeed.rValue;
				JSpeed.arrByte := TempJointVRev.q4;
				JointSpeed.q4 := JSpeed.rValue;
				JSpeed.arrByte := TempJointVRev.q5;
				JointSpeed.q5 := JSpeed.rValue;
				JSpeed.arrByte := TempJointVRev.q6;
				JointSpeed.q6 := JSpeed.rValue;
				
				Tool.arrByte := TempToolPosRev.q1;
				ToolPosition.q1 := Tool.rValue;
				Tool.arrByte := TempToolPosRev.q2;
				ToolPosition.q2 := Tool.rValue;
				Tool.arrByte := TempToolPosRev.q3;
				ToolPosition.q3 := Tool.rValue;
				Tool.arrByte := TempToolPosRev.q4;
				ToolPosition.q4 := RAD_TO_DEG(Tool.rValue);
				Tool.arrByte := TempToolPosRev.q5;
				ToolPosition.q5 := RAD_TO_DEG(Tool.rValue);
				Tool.arrByte := TempToolPosRev.q6;
				ToolPosition.q6 := RAD_TO_DEG(Tool.rValue);
				
				Delay_2(IN := TRUE, PT := T#0.5S);
				IF Delay_2.Q THEN
					Delay_2(IN := FALSE);
					RT_State := 3;
				END_IF
				
		3:	// Disconnect from RealTimePort
				Disconnect_RT(bExecute := TRUE);
							
				IF NOT Disconnect_RT.bBusy AND NOT Disconnect_RT.bError THEN
					Disconnect_RT.bExecute := FALSE;
					RT_State := 0;
				END_IF
		
	END_CASE
END_IF
//____________________________________________________________________________________________
// Zustandsmanagement

IF bFehler THEN 
	iState := 7;
END_IF

CASE iState OF 
	0: // AUS
		// DO
		
		// TRANSITION
			IF bEingeschalten THEN																	// Verbindung wird aufgebaut
				iState := 1;
			END_IF
			
	//____________________________________________________________________________________________
	1: // BEREIT
		// DO
			IF bStarten THEN
				bAmStarten := A_BewegungZuPosition();
			END_IF
			
			IF bAmStarten  THEN
				bAmStarten := FALSE;
				Delay_1(IN := TRUE, PT := T#0.2S);				 
			END_IF
			
			IF Delay_1.Q THEN
				Delay_1(IN := FALSE);
				bGestartet := TRUE;
			END_IF
		
		// TRANSITION
			IF bAusgeschalten THEN																	// Verbindung wird getrennt
				iState := 0;
			END_IF
			
																									// Manuell-Modus wird eingeschalten
													
			 IF bGestartet THEN																		// Objekt führt Prozessdurch
				 bGestartet := FALSE;
				 iState := 3;
			 END_IF			
	//____________________________________________________________________________________________
	2: // MANUELL
		// DO
		
		// TRANSITION
	
	//____________________________________________________________________________________________
	3: // LAUFEND
		// DO
			
			// Ermitteln von TargetPosition 
			IF NOT bSetvalues THEN
				// Kartesisch
				IF Prozessvariablen.MoveTyp = 0 OR Prozessvariablen.MoveTyp = 3 THEN
					// Absolut
					IF Prozessvariablen.PosTyp = 0 THEN
						TargetPosition.q1 := Prozessvariablen.q1;
						TargetPosition.q2 := Prozessvariablen.q2;
						TargetPosition.q3 := Prozessvariablen.q3;
						TargetPosition.q4 := Prozessvariablen.q4;
						TargetPosition.q5 := Prozessvariablen.q5;
						TargetPosition.q6 := Prozessvariablen.q6;		
					END_IF
										
					// Relativ
					IF Prozessvariablen.PosTyp = 1 THEN
						TargetPosition.q1 := ToolPosition.q1 + Prozessvariablen.q1;
						TargetPosition.q2 := ToolPosition.q2 + Prozessvariablen.q2;
						TargetPosition.q3 := ToolPosition.q3 + Prozessvariablen.q3;
						TargetPosition.q4 := ToolPosition.q4 + Prozessvariablen.q4;
						TargetPosition.q5 := ToolPosition.q5 + Prozessvariablen.q5;
						TargetPosition.q6 := ToolPosition.q6 + Prozessvariablen.q6;
					END_IF
					
				END_IF
				
				// Gelenkwinkel
				IF Prozessvariablen.MoveTyp = 1 THEN
					TargetPosition.q1 := Prozessvariablen.q1;
					TargetPosition.q2 := Prozessvariablen.q2;
					TargetPosition.q3 := Prozessvariablen.q3;
					TargetPosition.q4 := Prozessvariablen.q4;
					TargetPosition.q5 := Prozessvariablen.q5;
					TargetPosition.q6 := Prozessvariablen.q6;	
				END_IF
			
				bSetvalues := TRUE;
			END_IF

			// Vergleich zwischen IST und SOLL
			// Kartesisch
			IF Prozessvariablen.MoveTyp = 0 OR Prozessvariablen.MoveTyp = 3 THEN
				IF ABS(ABS(TargetPosition.q1) - ABS(ToolPosition.q1)) < 0.001 THEN
					bQ1 := TRUE;
				END_IF
				
				IF ABS(ABS(TargetPosition.q2) - ABS(ToolPosition.q2)) < 0.001 THEN
					bQ2 := TRUE;
				END_IF
				
				IF ABS(ABS(TargetPosition.q3) - ABS(ToolPosition.q3)) < 0.001 THEN
					bQ3 := TRUE;
				END_IF
				
				IF ABS(ABS(TargetPosition.q4) - ABS(ToolPosition.q4)) < 1 THEN
					bQ4 := TRUE;
				END_IF
				
				IF ABS(ABS(TargetPosition.q5) - ABS(ToolPosition.q5)) < 1 THEN
					bQ5 := TRUE;
				END_IF
				
				IF ABS(ABS(TargetPosition.q6) - ABS(ToolPosition.q6)) < 1 THEN
					bQ6 := TRUE;
				END_IF
			END_IF
			
			// Gelenkwinkel
			IF Prozessvariablen.MoveTyp = 1 THEN
				IF ABS(TargetPosition.q1) - ABS(JointPositions.q1) < 0.1 THEN
					bQ1 := TRUE;
				END_IF
				
				IF ABS(TargetPosition.q2) - ABS(JointPositions.q2) < 0.1 THEN
					bQ2 := TRUE;
				END_IF
				
				IF ABS(TargetPosition.q3) - ABS(JointPositions.q3) < 0.1 THEN
					bQ3 := TRUE;
				END_IF
				
				IF ABS(TargetPosition.q4) - ABS(JointPositions.q4) < 0.1 THEN
					bQ4 := TRUE;
				END_IF
				
				IF ABS(TargetPosition.q5) - ABS(JointPositions.q5) < 0.1 THEN
					bQ5 := TRUE;
				END_IF
				
				IF ABS(TargetPosition.q6) - ABS(JointPositions.q6) < 0.1 THEN
					bQ6 := TRUE;
				END_IF
			END_IF
			
			// Objekt schliessen Prozess ab
			IF bQ1 AND bQ2 AND bQ3 AND bQ4 AND bQ5 AND bQ6 THEN										// Abgeschlossener Prozess
				
				bQ1 := FALSE;
				bQ2 := FALSE;
				bQ3 := FALSE;
				bQ4 := FALSE;
				bQ5 := FALSE;
				bQ6 := FALSE;
				
				bObjektFertig := TRUE;
			END_IF
			
				
			// Objekt wird gestoppt durch Skill
			IF bSkillFertig THEN
				
				bQ1 := FALSE;
				bQ2 := FALSE;
				bQ3 := FALSE;
				bQ4 := FALSE;
				bQ5 := FALSE;
				bQ6 := FALSE;
				bSetvalues := FALSE;
				
				bBewegungStoppen := A_BewegungStoppen();
				
				IF bBewegungStoppen THEN
					bBewegungStoppen := FALSE;
					bAmStoppen := TRUE;
				END_IF
			END_IF 
			
			// Objekt wird gestoppt durch System
			IF bStoppen THEN
				
				bQ1 := FALSE;
				bQ2 := FALSE;
				bQ3 := FALSE;
				bQ4 := FALSE;
				bQ5 := FALSE;
				bQ6 := FALSE;
				bSetvalues := FALSE;
				
				bBewegungStoppen := A_BewegungStoppen();
				
				IF bBewegungStoppen THEN
					bBewegungStoppen := FALSE;
					bAmStoppen := TRUE;
				END_IF
			END_IF 
			
			// Stoppprozess
			IF bAmStoppen THEN
				IF JointSpeed.q1 < 0.001 THEN
					bVQ1 := TRUE;
				END_IF
				
				IF JointSpeed.q2 < 0.001 THEN
					bVQ2 := TRUE;
				END_IF
				
				IF JointSpeed.q3 < 0.001 THEN
					bVQ3 := TRUE;
				END_IF
				
				IF JointSpeed.q4 < 0.001 THEN
					bVQ4 := TRUE;
				END_IF
				
				IF JointSpeed.q5 < 0.001 THEN
					bVQ5 := TRUE;
				END_IF
				
				IF JointSpeed.q6 < 0.001 THEN
					bVQ6 := TRUE;
				END_IF
				
				IF bVQ1 AND bVQ2 AND bVQ3 AND bVQ4 AND bVQ5 AND bVQ6 THEN							// Gestoppter Prozess
					bVQ1 := FALSE;	
					bVQ2 := FALSE;	
					bVQ3 := FALSE;	
					bVQ4 := FALSE;	
					bVQ5 := FALSE;	
					bVQ6 := FALSE;	
					
					bAmStoppen := FALSE;
					bGestoppt := TRUE;
					
				END_IF
				
			END_IF
		
		// TRANSITION
			IF bObjektFertig THEN
				bObjektFertig := FALSE;
				bSetvalues := FALSE;
				iState := 4;
			END_IF
			
			IF bGestoppt THEN	
				bGestoppt := FALSE;	
				
				IF bSkillFertig THEN
					iState := 5;
				END_IF
					
				IF bStoppen THEN
					iState := 6;
				END_IF
					
			END_IF
	
	//____________________________________________________________________________________________
	4: // ABGESCHLOSSEN_INTERN
		// DO
		
		// TRANSITION
			IF bResettenSkill THEN																	// Objekt resetten		
				iState := 1;
			END_IF
	//____________________________________________________________________________________________
	5: // ABGESCHLOSSEN_EXTERN
		// DO																					
		
		// TRANSITION
			IF bResettenSkill THEN																	// Objekt resetten
				iState := 1;
			END_IF
	
	//____________________________________________________________________________________________
	6: // GESTOPPT
		// DO
		
		// TRANSITION
			IF bResettenSystem THEN																	// Objekt resetten
				iState := 1;
			END_IF
	
	//____________________________________________________________________________________________
	7: // FEHLER
		// DO
			bError := bFehler;
			
		// TRANSITION
			IF bResettenSystem THEN																	// Objekt resetten
				bFehler	 := FALSE;
				bError := FALSE;
				iState := 1;
			END_IF
	
END_CASE

METHOD A_BewegungStoppen : BOOL
VAR_INPUT
END_VAR
VAR
	stringFormat   		:FB_FormatString;		// Funktion für Stringerstellung	
	a					:INT := 2;

	Command				:T_MaxString;			// Commandstring
	CommandArray		:String_Array256;		// Byte-Array für Kommunikation mit Roboter
END_VAR
stringFormat(sFormat := 'stopj(%d)',
							arg1 := F_INT(a),
							bError => bError,
							nErrId => iErrorID,
							sOut => Command);	
							
// VOrbereiten von Array 
	CommandArray.sValue := Command;
	CommandArray.arrByte[LEN(CommandArray.sValue)] := 10;
	
// Senden von Array
	Send_STOP(cbLen := LEN(CommandArray.sValue),
			pSrc := ADR(CommandArray.arrByte),
			bExecute := TRUE);
			
	IF NOT Send_STOP.bBusy THEN
		Send_STOP(bExecute := FALSE);
		A_BewegungStoppen := TRUE;
	END_IF
END_METHOD

METHOD A_BewegungZuPosition : BOOL
VAR 
	
	x					:LREAL;				// X-Koordinate
	y					:LREAL;				// Y-Koordinate
	z					:LREAL;				// Z-Koordinate
	rx					:LREAL;				// Orintierung um X-Achse
	ry					:LREAL;				// Orientierung um Y-Achse
	rz					:LREAL;				// Orientierung um Z-Achse
	
	q1					:LREAL;				// Joint-Position 1
	q2					:LREAL;				// Joint-Position 2
	q3					:LREAL;				// Joint-Position 3
	q4					:LREAL;				// Joint-Position 4
	q5					:LREAL;				// Joint-Position 5
	q6					:LREAL;				// Joint-Position 6

	stringFormat   : FB_FormatString;		// Funktion für Stringerstellung

	pose			:T_MaxString;			// Positionsstring
	Command			:T_MaxString;			// Commandstring
	
	CommandArray	:String_Array256;			// Byte-Array für Kommunikation mit Roboter
	
END_VAR
VAR_INPUT
	
END_VAR
// Einfluss von Positionart
	IF Prozessvariablen.PosTyp = 1 THEN		// Relative Bewegung
		
		x := ToolPosition.q1 + Prozessvariablen.q1;
		y := ToolPosition.q2 + Prozessvariablen.q2;
		z := ToolPosition.q3 + Prozessvariablen.q3;
		rx := DEG_TO_RAD(ToolPosition.q4 + Prozessvariablen.q4);
		ry := DEG_TO_RAD(ToolPosition.q5 + Prozessvariablen.q5);
		rz := DEG_TO_RAD(ToolPosition.q6 + Prozessvariablen.q6);
		
	END_IF
	
	IF Prozessvariablen.PosTyp = 0 THEN		// Absolute Bewegung
		
		x := Prozessvariablen.q1;
		y := Prozessvariablen.q2;
		z := Prozessvariablen.q3;
		rx := DEG_TO_RAD(Prozessvariablen.q4);
		ry := DEG_TO_RAD(Prozessvariablen.q5);
		rz := DEG_TO_RAD(Prozessvariablen.q6);
		
	END_IF
	
	stringFormat(sFormat := 'p[%.3f,%.3f,%.3f,%.3f,%.3f,%.3f]',
			arg1 := F_LREAL(x),
			arg2 := F_LREAL(y),
			arg3 := F_LREAL(z),
			arg4 := F_LREAL(rx),
			arg5 := F_LREAL(ry),
			arg6 := F_LREAL(rz),
			bError => bError,
			nErrId => iErrorID,
			sOut => pose);

// Einlfuss von Bewegungsart
	IF Prozessvariablen.MoveTyp = 0 THEN			// Move to position (linear in tool-space)
													// movel(pose, a=1.2, v=0.25, t=0, r=0)
		stringFormat(sFormat := 'movel(%s, a=%.2f, v=%.2f)',
							arg1 := F_STRING(pose),
							arg2 := F_LREAL(Prozessvariablen.a),
							arg3 := F_LREAL(Prozessvariablen.v),
							bError => bError,
							nErrId => iErrorID,
							sOut => Command);											
	END_IF
	
	IF Prozessvariablen.MoveTyp = 1 THEN			// Move to position (linear in joint-space)
													// movej(q, a=1.4, v=1.05, t=0, r =0)
		q1 := DEG_TO_RAD(Prozessvariablen.q4);
		q2 := DEG_TO_RAD(Prozessvariablen.q5);
		q3 := DEG_TO_RAD(Prozessvariablen.q6);
		q4 := DEG_TO_RAD(Prozessvariablen.q4);
		q5 := DEG_TO_RAD(Prozessvariablen.q5);
		q6 := DEG_TO_RAD(Prozessvariablen.q6);
		
		stringFormat(sFormat := 'movej([%.3f,%.3f,%.3f,%.3f,%.3f,%.3f], a=%.2f, v=%.2f)',
							arg1 := F_LREAL(q1),
							arg2 := F_LREAL(q2),
							arg3 := F_LREAL(q3),
							arg4 := F_LREAL(q4),
							arg5 := F_LREAL(q5),
							arg6 := F_LREAL(q6),
							arg7 := F_LREAL(Prozessvariablen.a),
							arg8 := F_LREAL(Prozessvariablen.v),
							bError => bError,
							nErrId => iErrorID,
							sOut => Command);	
													
	END_IF
	
	IF Prozessvariablen.MoveTyp = 2 THEN			// Move Circular: Move to position (circular in tool-space)
													//movec(pose_via, pose_to, a=1.2, v=0.25, r =0, mode=0)
													
		
	END_IF
	
	IF Prozessvariablen.MoveTyp = 3 THEN			// Move Process
													// movep(pose, a=1.2, v=0.25, r=0)
		stringFormat(sFormat := 'movep(%s, a=%.2f, v=%.2f)',
							arg1 := F_STRING(pose),
							arg2 := F_LREAL(Prozessvariablen.a),
							arg3 := F_LREAL(Prozessvariablen.v),
							bError => bError,
							nErrId => iErrorID,
							sOut => Command);												
	END_IF

// Vorbereiten von Array
	CommandArray.sValue := Command;
	CommandArray.arrByte[LEN(CommandArray.sValue)] := 10;

// Senden von Array	
	Send_START(cbLen := LEN(CommandArray.sValue),
			pSrc := ADR(CommandArray.arrByte),
			bExecute := TRUE);
			
	IF NOT Send_START.bBusy THEN
		Send_START(bExecute := FALSE);
		A_BewegungZuPosition := TRUE;
	END_IF
END_METHOD

PROPERTY P_JointPosition : sPositionValues
GET
P_JointPosition := JointPositions;
END_GET
END_PROPERTY

PROPERTY P_ToolPosition : sPositionValues
GET
P_ToolPosition := ToolPosition;
END_GET
END_PROPERTY

METHOD Trennen : BOOL
VAR_INPUT
END_VAR
// Ausführen von Funktionalitäten
	Disconnect(sSrvNetId := sSrvNetId,
			bExecute := TRUE,
			tTimeout := tTimeout,
			bError => bError,
			nErrId => iErrorID);
	
	IF NOT Disconnect.bBusy AND NOT bError THEN
		Trennen := TRUE;
		Disconnect(bExecute := FALSE);
	END_IF
END_METHOD

METHOD Verbinden : BOOL 
VAR
	
END_VAR
// Ausführen von Funktionalitäten
	Connect(sSrvNetId := sSrvNetId,
			sRemoteHost := sIP,
			nRemotePort := iPort_Prim,
			bExecute := TRUE,
			tTimeout := tTimeout,
			bError => bError,
			nErrId => iErrorID,
			hSocket => hSocket);
			
	IF hSocket.handle <> 0 THEN
		Verbinden := TRUE;
		Connect(bExecute := FALSE);
		Connect_RT(bExecute := FALSE);
	END_IF
END_METHOD

END_FUNCTION_BLOCK

// ---- POUs/02_Anlagenmodell/01_Grundstruktur/GrundstrukturObjekt.TcPOU
FUNCTION_BLOCK GrundstrukturObjekt IMPLEMENTS I_State_Object
VAR_INPUT
	bReset				:BOOL;				// Resett für den Manuell-Modus
	iMode				:INT;				// Information über aktuellen Betriebsmodi 
	iSysState			:eSystemState;		// Information über Stand von System
	iSysCommand		  	:eSystemCommand;	// Steuerungsvariabel von System
	iSkillCommand_1 	:eSkillCommand;		// Steuerungsvariabel von Skill_1
END_VAR
VAR_OUTPUT
	bError				:BOOL;				// Information ob sich Objekt in Fehlerzustand befindet
	iErrorID			:UDINT;				// Information um welchen Fehler es sich handelt	
END_VAR
VAR
	iState				:eObjectAktorState;		// Information über Zustand von Skill
	
	// Zustandsvariablen
	bEinschalten			:BOOL;			// Objekt einschalten
	bAusschalten			:BOOL;			// Objekt ausschalten
 	bStarten				:BOOL;			// Objekt starten
	bObjektFertig			:BOOL;			// Objekt hat Prozess abgeschlossen
	bSkillFertig			:BOOL;			// Skill hat Prozess abgeschlossen
	bStoppen				:BOOL;			// Objekt wurde gestoppt
	bResettenSkill			:BOOL;			// Das Objekt wird durch den Skill resettet
	bResettenSystem			:BOOL;			// Das Objekt wird durch das System resettet 
	bFehler					:BOOL;			// Das Objket hat einen Fehler
	
	iFehlerID				:UDINT;


	
	
	
END_VAR

PROPERTY P_State : eObjectAktorState
GET
P_State := iState;
END_GET
END_PROPERTY

END_FUNCTION_BLOCK

// ---- POUs/02_Anlagenmodell/02_Objektklassen/FB_SmartGreifer.TcPOU
FUNCTION_BLOCK FB_SmartGreifer EXTENDS GrundstrukturObjekt
VAR_INPUT
	iSkillCommand_2			:eSkillCommand;		// Steuerungsvariabel von Skill_2
	iSkillCommand_3			:eSkillCommand;		// Steuerungsvariabel von Skill_2
	iSkillCommand_4			:eSkillCommand;		// Steuerungsvariabel von Skill_2
	Prozessvariablen		:sSmartGreiferProzessVariablen; 
END_VAR
VAR_OUTPUT
END_VAR
VAR
	// Instanziierung von Kommunikationsbausteine 
	Communication			:ModbusRtuMasterV2_KL6x22B;
	
	// Kommunikationsvariablen
	UnitID      			:BYTE := 9;
    Quantity    			:WORD;
    MBAddr      			:WORD;
	Timeout     			:TIME := T#5S;
	cbRead					:UINT;
	DataSend				:ARRAY[0..5] OF BYTE;
	DataRead				:ARRAY[0..5] OF BYTE;
	
	// Managementvariablen
	iStartUp			:INT;
	iProzess			:INT;
	iSkillOption		:INT;
	
	bGreiferReset		:BOOL;
	bGreiferLesen		:BOOL;
	
	bAmEinschalten		:BOOL;
	bEingeschalten		:BOOL;
	
	bGestartet			:BOOL;
	
	
	CheckTimer			:TON;
	Delay				:TON;
	
	// Prozessvariablen
	iPos				:BYTE;
	iGeschw				:BYTE;
	iKraft				:BYTE;
	
	// Eigenschaftsvariablen
	iPosMax				:REAL := 85;
	iGeschwMin			:REAL := 20;
	iGeschwMax			:REAL := 150;
	iKraftMin			:REAL := 20;
	iKraftMax			:REAL := 235;
	Anschlag			:BYTE;

	
	
	
END_VAR

// Instanziierungen	
Communication(
	UnitID 		:= UnitID,
	Timeout 	:= Timeout,
	Error 		=> bError,
	ErrorId 	=> iErrorID,
	cbRead 		=> cbRead);


//____________________________________________________________________________________________
// Input-Command-Verwaltung
	// System
	IF iSysCommand = 2 AND iState = 0 THEN			// Objekt einschalten
		bEinschalten := TRUE;
	ELSE 
		bEinschalten := FALSE;
	END_IF
	
	IF iSysCommand = 1 AND iState = 1 THEN				// Objekt ausschalten
		bAusschalten := TRUE;		
	ELSE 
		bAusschalten := FALSE;		
	END_IF
	
	IF iSysCommand = 3 THEN								// Objekt beendet Prozess
		bStoppen := TRUE;
	ELSE
		bStoppen := FALSE;
	END_IF
	
	IF iSysCommand = 4 THEN								// System resettet Objekt
		bResettenSystem := TRUE;
	ELSE
		bResettenSystem := FALSE;
	END_IF
	
	// Skill
	IF iSkillCommand_1 = 1 OR iSkillCommand_2 = 1 OR  iSkillCommand_3 = 1 OR iSkillCommand_4 = 1 THEN	// Skill startet Prozess
		IF iSkillCommand_1 = 1 THEN
			iSkillOption := 1;
		END_IF
		
		IF iSkillCommand_2 = 1 THEN
			iSkillOption := 2;
		END_IF
		
		IF iSkillCommand_3 = 1 THEN
			iSkillOption := 3;
		END_IF
		
		IF iSkillCommand_4 = 1 THEN
			iSkillOption := 4;
		END_IF
		
		bStarten := TRUE;
	ELSE 
		bStarten := FALSE;
	END_IF
	
	IF iSkillCommand_1 = 2 OR iSkillCommand_2 = 2 THEN	// Skill beendet Prozess
		bSkillFertig := TRUE;
	ELSE
		bSkillFertig := FALSE;
	END_IF
	
	IF iSkillCommand_1 = 3 OR iSkillCommand_2 = 3 THEN	// Skill resettet Objekt
 		bResettenSkill := TRUE;
	ELSE
		bResettenSkill := FALSE;
	END_IF

//____________________________________________________________________________________________
// Interner Methodenaufruf (Durch System oder Skill)

//____________________________________________________________________________________________
// Datenerfassungsprozess

//____________________________________________________________________________________________
// Zustandsmanagement

IF bFehler THEN 
	iState := 7;
END_IF

CASE iState OF 
	0: // AUS
		// DO
		IF bEinschalten THEN
			CASE iStartUP OF
				0: // Greifer Resetten
					bGreiferReset := Resetten();
					
					IF bGreiferReset THEN
						bGreiferReset := FALSE;
						iStartUp := 1;
					END_IF
				1: // Greifer Aktivieren
					bAmEinschalten := Aktivieren();
					
					IF bAmEinschalten THEN 
						bAmEinschalten := FALSE;
						Delay(IN:= TRUE, PT := T#1S);
					END_IF
					
					IF Delay.Q THEN
						Delay(IN:= FALSE);
						iStartUp := 2;
					END_IF
					
				2:
					bGreiferLesen := StatusLesen(NrOfReg := 1);
					
					IF bGreiferLesen THEN
						bGreiferLesen := FALSE;
						IF DataRead[1] = 49  AND DataRead[0] = 0 THEN
							bEingeschalten := TRUE;
						END_IF
					END_IF
			END_CASE
		END_IF
		
		// TRANSITION
		IF bEingeschalten THEN																			// Verbindung wird aufgebaut
			bEingeschalten := FALSE;
			iStartUp := 0;
			iState := 1;
		END_IF
			
	//____________________________________________________________________________________________
	1: // BEREIT
		// DO
			Anschlag := 0;

		// TRANSITION		
			IF bAusschalten THEN
				iState := 0;
			END_IF
																									// Manuell-Modus wird eingeschalten
													
			 IF bStarten THEN																		// Objekt führt Prozessdurch
				 iState := 3;
			 END_IF			
	//____________________________________________________________________________________________
	2: // MANUELL
		// DO
		
		// TRANSITION
	
	//____________________________________________________________________________________________
	3: // LAUFEND
		// DO
			
			// Aktionsprozess 
			CASE iSkillOption OF 
				1:	// Definierte Position anfahren
					CASE iProzess OF 
					0: // Aktion durchführen
						iPos := REAL_TO_BYTE((255.00/iPosMax) *  (iPosMax - Prozessvariablen.Pos));	
						iGeschw := REAL_TO_BYTE((255.00 / 100.00) * Prozessvariablen.Geschw );
						iKraft := REAL_TO_BYTE((255.00 / 100.00) * Prozessvariablen.F);
					
						bGestartet := A_PositionAnfahren(iPos := iPos, iGeschw := iGeschw, iKraft := iKraft);
						
						IF bGestartet THEN
							bGestartet := FALSE;
							Delay(IN:= TRUE, PT := T#1S);
						END_IF
						
						IF Delay.Q THEN
							Delay(IN:= FALSE);
							iProzess := 1;
						END_IF
					
					1: // Prüfen ob Aktion erledigt 
						bGreiferLesen := StatusLesen(NrOfReg := 3);
						CheckTimer(IN := TRUE, PT := T#5S);
						
						IF bGreiferLesen THEN
							bGreiferLesen := FALSE;
							
							// Greifer hat Position erreicht
							IF 	DataRead[0] = 0 		AND
								DataRead[1] = 249 		AND
								DataRead[2] = iPos 		AND
								DataRead[3] = 0 		AND
								DataRead[4] = 0 		AND
								DataRead[5] = iPos		THEN
								
								CheckTimer(IN := FALSE);
								iProzess := 0;
								bObjektFertig := TRUE;
							END_IF
							
							// Greifer ist in Hinderniss gefahren
							IF 	DataRead[0] = 0 		AND
								DataRead[1] = 185 		AND
								DataRead[3] = 0 		AND
								DataRead[4] = 0 		THEN
								
								CheckTimer(IN := FALSE);
								iProzess := 0;
								bFehler := TRUE;
								iFehlerID := 202;
							END_IF
							
						END_IF
						
						// Zeit wurde überschritten
						IF CheckTimer.Q THEN		
							iProzess := 0;
							CheckTimer(IN := FALSE);
							bFehler := TRUE;
							iFehlerID := 201;
						END_IF
					END_CASE
					
				//______________________________________________________________________________________________________	
				2:	// Greifabstand ermitteln
					CASE iProzess OF 
					0: // Aktion durchführen
						iPos := REAL_TO_BYTE(((255/iPosMax) * (iPosMax - Prozessvariablen.Pos)));	
						iGeschw := REAL_TO_BYTE((255.00 / 100.00) * Prozessvariablen.Geschw );
						iKraft := REAL_TO_BYTE((255.00 / 100.00) * Prozessvariablen.F);
					
						bGestartet := A_PositionAnfahren(iPos := iPos, iGeschw := iGeschw, iKraft := iKraft);
						
						IF bGestartet THEN
							bGestartet := FALSE;
							Delay(IN:= TRUE, PT := T#1S);
						END_IF
						
						IF Delay.Q THEN
							Delay(IN:= FALSE);
							iProzess := 1;
						END_IF
					
					1: // Prüfen ob Aktion erledigt 
						bGreiferLesen := StatusLesen(NrOfReg := 3);
						CheckTimer(IN := TRUE, PT := T#5S);
						
						IF bGreiferLesen THEN
							bGreiferLesen := FALSE;
							
							// Greifer hat Position erreicht
							IF 	DataRead[0] = 0 		AND
								DataRead[1] = 249 		AND
								DataRead[2] = iPos 		AND
								DataRead[3] = 0 		AND
								DataRead[4] = 0 		AND
								DataRead[5] = iPos		THEN
								
								CheckTimer(IN := FALSE);
								Anschlag := iPos;
								iProzess := 0;
								bObjektFertig := TRUE;
							END_IF
							
							// Greifer ist in Hinderniss gefahren
							IF 	DataRead[0] = 0 		AND
								DataRead[1] = 185 		AND
								DataRead[3] = 0 		AND
								DataRead[4] = 0 		THEN
								
								Anschlag := DataRead[5];
								CheckTimer(IN := FALSE);
								iProzess := 0;
								bObjektFertig := TRUE;								
							END_IF
							
						END_IF
						
						// Zeit wurde überschritten
						IF CheckTimer.Q THEN		
							iProzess := 0;
							CheckTimer(IN := FALSE);
							bFehler := TRUE;
							iFehlerID := 201;
						END_IF
					END_CASE
				
				//______________________________________________________________________________________________________	
				3:	// Grifer komplett schliessen
					CASE iProzess OF 
					0: // Aktion durchführen
						iPos := 200;	
						iGeschw := 100;
						iKraft := 0;
						
							bGestartet := A_PositionAnfahren(iPos := iPos, iGeschw := iGeschw, iKraft := iKraft);
					
						IF bGestartet THEN
							bGestartet := FALSE;
							Delay(IN:= TRUE, PT := T#1S);
						END_IF
						
						IF Delay.Q THEN
							Delay(IN:= FALSE);
							iProzess := 1;
						END_IF
					
					1: // Prüfen ob Aktion erledigt 
						bGreiferLesen := StatusLesen(NrOfReg := 3);
						CheckTimer(IN := TRUE, PT := T#5S);
						
						IF bGreiferLesen THEN
							bGreiferLesen := FALSE;
							
							// Greifer ist in Hinderniss gefahren
							IF 	DataRead[0] = 0 		AND
								DataRead[1] = 249 		AND
								DataRead[3] = 0 		AND
								DataRead[4] = 0 		THEN
								
								CheckTimer(IN := FALSE);
								iProzess := 0;
								bObjektFertig := TRUE;								
							END_IF
							
						END_IF
						
						// Zeit wurde überschritten
						IF CheckTimer.Q THEN		
							iProzess := 0;
							CheckTimer(IN := FALSE);
							bFehler := TRUE;
							iFehlerID := 201;
						END_IF
					END_CASE
					
				//______________________________________________________________________________________________________
				4: 	// Greifer komplett öffnen
					CASE iProzess OF 
					0: // Aktion durchführen
						iPos := 0;	
						iGeschw := 100;
						iKraft := 100;
						
						bGestartet := A_PositionAnfahren(iPos := iPos, iGeschw := iGeschw, iKraft := iKraft);
		
						
						IF bGestartet THEN
							bGestartet := FALSE;
							Delay(IN:= TRUE, PT := T#1S);
						END_IF
						
						IF Delay.Q THEN
							Delay(IN:= FALSE);
							iProzess := 1;
						END_IF
					
					
					1: // Prüfen ob Aktion erledigt 
						bGreiferLesen := StatusLesen(NrOfReg := 3);
						
						CheckTimer(IN := TRUE, PT := T#5S);
						
						IF bGreiferLesen THEN
							bGreiferLesen := FALSE;
							
							// Greifer hat Position erreicht
							IF 	DataRead[0] = 0 		AND
								DataRead[1] = 249 		AND
								DataRead[2] = 0 		AND
								DataRead[3] = 0 		AND
								DataRead[4] = 0 		THEN
								
								CheckTimer(IN := FALSE);
								iProzess := 0;
								bObjektFertig := TRUE;
							END_IF
							
							// Greifer ist in Hinderniss gefahren
							IF 	DataRead[0] = 0 		AND
								DataRead[1] = 185 		AND
								DataRead[3] = 0 		AND
								DataRead[4] = 0 		THEN
								
								CheckTimer(IN := FALSE);
								iProzess := 0;
								bFehler := TRUE;
								iFehlerID := 202;
							END_IF
					
							
						END_IF
						
						// Zeit wurde überschritten
						IF CheckTimer.Q THEN		
							iProzess := 0;
							CheckTimer(IN := FALSE);
							bFehler := TRUE;
							iFehlerID := 201;
						END_IF
					END_CASE
			END_CASE			
		
		// TRANSITION
			IF bObjektFertig THEN
				bObjektFertig := FALSE;
				iState := 4;
			END_IF
			
			IF bStoppen THEN	
				
				IF bSkillFertig THEN
					iState := 5;
				END_IF
					
				IF bStoppen THEN
					iState := 6;
				END_IF
					
			END_IF
	
	//____________________________________________________________________________________________
	4: // ABGESCHLOSSEN_INTERN
		// DO
		
		// TRANSITION
			IF bResettenSkill THEN																	// Objekt resetten		
				iState := 1;
			END_IF
	//____________________________________________________________________________________________
	5: // ABGESCHLOSSEN_EXTERN
		// DO																					
		
		// TRANSITION
			IF bResettenSkill THEN																	// Objekt resetten
				iState := 1;
			END_IF
	
	//____________________________________________________________________________________________
	6: // GESTOPPT
		// DO
		
		// TRANSITION
			IF bResettenSystem THEN																	// Objekt resetten
				iState := 1;
			END_IF
	
	//____________________________________________________________________________________________
	7: // FEHLER
		// DO
			bError := bFehler;
			iErrorID := iFehlerID;
			
		// TRANSITION
			IF bResettenSystem THEN																	// Objekt resetten
				bFehler	 := FALSE;
				bError := FALSE;
				iErrorID := 0;
				iState := 1;
			END_IF
	
END_CASE

METHOD A_PositionAnfahren : BOOL
VAR_INPUT
	iPos		:BYTE;
	iGeschw		:BYTE;
	iKraft		:BYTE;
END_VAR
// Definieren der Anzahl von Daten-Bytes 
Quantity := 3;

// Definieren von Register
MBAddr := 1000;

// Definieren der Daten
DataSend[0] := 0;
DataSend[1] := 9;
DataSend[2] := iPos;
DataSend[3] := 0;
DataSend[4] := iKraft;
DataSend[5] := iGeschw;

// Senden von Daten an entsprechendes Register
Communication.WriteRegs(
	Quantity 	:= Quantity,
	MBAddr 		:= MBAddr,
	cbLength 	:= SIZEOF(DataSend),
	pMemoryAddr := ADR(DataSend),
	Execute 	:= TRUE);
	
IF NOT Communication.BUSY THEN
	Communication.WriteRegs(Execute := FALSE);
	A_PositionAnfahren := TRUE;
END_IF
END_METHOD

METHOD Aktivieren : BOOL
VAR_INPUT
END_VAR
// Definieren der Anzahl von Daten-Bytes 
Quantity := 3;

// Definieren von Register
MBAddr := 1000;

// Definieren der Daten
DataSend[0] := 0;
DataSend[1] := 1;
DataSend[2] := 0;
DataSend[3] := 0;
DataSend[4] := 0;
DataSend[5] := 0;

// Senden von Daten an entsprechendes Register
Communication.WriteRegs(
	Quantity 	:= Quantity,
	MBAddr 		:= MBAddr,
	cbLength 	:= SIZEOF(DataSend),
	pMemoryAddr := ADR(DataSend),
	Execute 	:= TRUE);
	
IF NOT Communication.BUSY THEN
	Communication.WriteRegs(Execute := FALSE);
	Aktivieren := TRUE;
END_IF
END_METHOD

PROPERTY AnschlagPos : BYTE
GET
AnschlagPos := Anschlag;
END_GET
END_PROPERTY

METHOD Resetten : BOOL
VAR_INPUT
END_VAR
// Definieren der Anzahl von Daten-Bytes 
Quantity := 3;

// Definieren von Register
MBAddr := 1000;

// Definieren der Daten
DataSend[0] := 0;
DataSend[1] := 0;
DataSend[2] := 0;
DataSend[3] := 0;
DataSend[4] := 0;
DataSend[5] := 0;

// Senden von Daten an entsprechendes Register
Communication.WriteRegs(
	Quantity 	:= Quantity,
	MBAddr 		:= MBAddr,
	cbLength 	:= SIZEOF(DataSend),
	pMemoryAddr := ADR(DataSend),
	Execute 	:= TRUE);
	
IF NOT Communication.BUSY THEN
	Communication.WriteRegs(Execute := FALSE);
	Resetten := TRUE;
END_IF
END_METHOD

METHOD StatusLesen : BOOL
VAR_INPUT
	NrOfReg			:WORD;
END_VAR
// Definieren von Register
MBAddr := 2000;


// Lesen von Daten des entsprechenden Registers
Communication.ReadRegs(
	Quantity 	:= NrOfReg,
	MBAddr 		:= MBAddr,
	cbLength 	:= SIZEOF(DataRead),
	pMemoryAddr := ADR(DataRead),
	Execute 	:= TRUE);
	
	
IF NOT Communication.BUSY THEN
	Communication.ReadRegs(Execute := FALSE);
	StatusLesen := TRUE;
END_IF
END_METHOD

END_FUNCTION_BLOCK

// ---- POUs/02_Anlagenmodell/02_Objektklassen/FB_Kraftsensor.TcPOU
FUNCTION_BLOCK FB_Kraftsensor EXTENDS GrundstrukturObjekt
VAR_INPUT
	
	// Kommunikationsvariablen
	sIP					:T_IPv4Addr;
	iPort				:UINT;
	
END_VAR
VAR_OUTPUT
END_VAR
VAR
	// Instanziierung von Kommunikationsbausteine
	Connect				:FB_SocketConnect;
	Disconnect			:FB_SocketClose;
	Send				:FB_SocketSend;
	Receive				:FB_SocketReceive;
	
	// Kommunikationsvariablen
	sSrvNetId   		:T_AmsNetId := '';
	tTimeout    		:TIME := T#45S;(*!!!*)
	hSocket    			:T_HSOCKET;
	
	// RealTimeDatenerfassung
	RT_State			:INT;							// RealTime-State-Variable
	{attribute 'TcSwapWord'}
	SendData 			:Request;
	{attribute 'TcSwapWord'}
	ReceivedData		:Response_Values;				// Erhaltene Daten von Roboter
	nRecBytes			:UDINT;							// Anzahl der erhaltenen Bytes
	
	CPF					:INT := 10000;					// Counts per Force value
	CPT					:INT := 10000;					// Counts per Torque value (Noch mal 10 rechnen)
	ScalefactorFx		:INT := 200;					// Additional scaling factor (for the Fx,Fy,Fz,Tx,Ty,Tz)
	ScalefactorFy		:INT := 200;					// Additional scaling factor (for the Fx,Fy,Fz,Tx,Ty,Tz)
	ScalefactorFz		:INT := 200;					// Additional scaling factor (for the Fx,Fy,Fz,Tx,Ty,Tz)
	ScalefactorTx		:INT := 100;					// Additional scaling factor (for the Fx,Fy,Fz,Tx,Ty,Tz)
	ScalefactorTy		:INT := 100;					// Additional scaling factor (for the Fx,Fy,Fz,Tx,Ty,Tz)
	ScalefactorTz		:INT := 65;						// Additional scaling factor (for the Fx,Fy,Fz,Tx,Ty,Tz)
	
	RohArray			:Int_2Byte;
	SwitchArray			:ARRAY[0..1] OF BYTE;
	SwichValue			:Array2_Int;
		
	Rohdaten			:Kraftvariablen;				// Rohwerte der Messung 
	Messung				:Kraftvariablen;				// Werte in Newton / Newtonmeter 

	// Managementvariablen
	bAusgeschalten		:BOOL;
	bManOn				:BOOL;
	m					:INT;
	
	// Eigenschaftsmethoden
	sLimitGrenze		:sKraftVariablen;
	sErreichtGrenze		:sKraftVariablen;
	bLimit				:BOOL;
	bLimitx				:BOOL;
	bLimity				:BOOL;
	bLimitz				:BOOL;
	bErreicht			:BOOL;
	bErreichtx			:BOOL;
	bErreichty			:BOOL;
	bErreichtz			:BOOL;
	
END_VAR

// Instanziierungen
Connect(sSrvNetId := sSrvNetId,
		sRemoteHost := sIP,
		nRemotePort := iPort,
		tTimeout := tTimeout,
		bError => bError,
		nErrId => iErrorID,
		hSocket => hSocket);	
						
Send(sSrvNetId := sSrvNetId,
		hSocket := hSocket,
		tTimeout := tTimeout,
		cbLen := SIZEOF(SendData),
		pSrc := ADR(SendData),
		bError => bError,
		nErrId => iErrorID);
						
Receive(sSrvNetId := sSrvNetId,
		hSocket := hSocket,
		cbLen := SIZEOF(ReceivedData),
		pDest := ADR(ReceivedData),
		tTimeout := tTimeout,
		bError => bError,
		nErrId => iErrorID,
		nRecBytes => nRecBytes);
						
Disconnect(sSrvNetId := sSrvNetId,
			hSocket := hSocket,
			tTimeout := tTimeout,
			bError => bError,
			nErrId => iErrorID);
	
//____________________________________________________________________________________________
// Input-Command-Verwaltung
	// System
	IF iSysCommand = 2 AND iState = 0 THEN			// Objekt einschalten
		bEinschalten := TRUE;
	ELSE 
		bEinschalten := FALSE;
	END_IF
	
	IF iSysCommand = 1 AND iState = 1 THEN			// Objekt ausschalten
		bAusschalten := TRUE;		
	ELSE 
		bAusschalten := FALSE;		
	END_IF
	
	IF iSysCommand = 3 THEN							// Objekt beendet Prozess
		bStoppen := TRUE;
	ELSE
		bStoppen := FALSE;
	END_IF
	
	IF iSysCommand = 4 THEN							// System resettet Objekt
		bResettenSystem := TRUE;
	ELSE
		bResettenSystem := FALSE;
	END_IF
	
	// Skill
	IF iSysState = 1 THEN						// Skill startet Prozess
		bStarten := TRUE;
	ELSE 
		bStarten := FALSE;
	END_IF
	
	IF iSkillCommand_1 = 2 THEN						// Skill beendet Prozess
		bSkillFertig := TRUE;
	ELSE
		bSkillFertig := FALSE;
	END_IF
	
	IF iSkillCommand_1 = 3 THEN						// Skill resettet Objekt
 		bResettenSkill := TRUE;
	ELSE
		bResettenSkill := FALSE;
	END_IF

//____________________________________________________________________________________________
// Interner Methodenaufruf (Durch System oder Skill)

//____________________________________________________________________________________________
// Datenerfassungsprozess
IF bManOn OR iState = 3 THEN
	CASE RT_State OF 
		0:	// Connect to RealTimePort
				Connect(bExecute := TRUE);			
					
				IF NOT Connect.bBusy AND NOT Connect.bError THEN
					Connect.bExecute := FALSE;
					RT_State := 1;
				END_IF
				
		1: 	// Send Data 
					SendData.Command := 0;
					Send(bExecute := TRUE);
				
					IF NOT Send.bBusy AND NOT Send.bError THEN
						Send.bExecute := FALSE;
						RT_State := 2;
					END_IF
		
		2:	// Get Data 
				Receive(bExecute := TRUE);
			
				IF NOT Receive.bBusy AND NOT Receive.bError THEN
					Receive.bExecute := FALSE;
					RT_State := 3;
				END_IF
				
		3:	// Convert Data
		
			RohArray.sValue := ReceivedData.Fx;
			SwitchArray[0] := RohArray.arrByte[1];
			SwitchArray[1] := RohArray.arrByte[0];
			SwichValue.arrByte := SwitchArray;
			Rohdaten.Fx := SwichValue.sValue;
			Messung.Fx := Rohdaten.Fx * ScalefactorFx / (CPF);
			
			RohArray.sValue := ReceivedData.Fy;
			SwitchArray[0] := RohArray.arrByte[1];
			SwitchArray[1] := RohArray.arrByte[0];
			SwichValue.arrByte := SwitchArray;
			Rohdaten.Fy := SwichValue.sValue;
			Messung.Fy := Rohdaten.Fy * ScalefactorFy / (CPF);
			
			RohArray.sValue := ReceivedData.Fz;
			SwitchArray[0] := RohArray.arrByte[1];
			SwitchArray[1] := RohArray.arrByte[0];
			SwichValue.arrByte := SwitchArray;
			Rohdaten.Fz := SwichValue.sValue;
			Messung.Fz := Rohdaten.Fz * ScalefactorFz / (CPF);
			
			RohArray.sValue := ReceivedData.Tx;
			SwitchArray[0] := RohArray.arrByte[1];
			SwitchArray[1] := RohArray.arrByte[0];
			SwichValue.arrByte := SwitchArray;
			Rohdaten.Tx := SwichValue.sValue;
			Messung.Tx := Rohdaten.Tx * ScalefactorTx / (CPT);
			
			RohArray.sValue := ReceivedData.Ty;
			SwitchArray[0] := RohArray.arrByte[1];
			SwitchArray[1] := RohArray.arrByte[0];
			SwichValue.arrByte := SwitchArray;
			Rohdaten.Ty := SwichValue.sValue;
			Messung.Ty := Rohdaten.Ty * ScalefactorTy / (CPT);
			
			RohArray.sValue := ReceivedData.Tz;
			SwitchArray[0] := RohArray.arrByte[1];
			SwitchArray[1] := RohArray.arrByte[0];
			SwichValue.arrByte := SwitchArray;
			Rohdaten.Tz := SwichValue.sValue;
			Messung.Tz := Rohdaten.Tz * ScalefactorTz / (CPT);
			
		
			RT_State := 4;
				
		4:	// Disconnect from RealTimePort
				Disconnect(bExecute := TRUE);
							
				IF NOT Disconnect.bBusy AND NOT Disconnect.bError THEN
					Disconnect.bExecute := FALSE;
					RT_State := 0;
				END_IF
		
	END_CASE
END_IF

//____________________________________________________________________________________________
// Zustandsmanagement

IF bFehler THEN 
	iState := 7;
END_IF

CASE iState OF 
	0: // AUS
		// DO
		
		// TRANSITION
			IF bEinschalten THEN																	// Verbindung wird aufgebaut
				iState := 1;
			END_IF
			
	//____________________________________________________________________________________________
	1: // BEREIT
		// DO
			IF bAusschalten THEN																	// Objekt ausschalten	
				Disconnect(bExecute := TRUE);
				IF NOT Disconnect.bBusy AND NOT Disconnect.bError THEN
					Disconnect.bExecute := FALSE;
					bAusgeschalten := TRUE;
				END_IF	
				
			END_IF

		// TRANSITION
			IF bAusgeschalten THEN																	// Objekt ausschalten
				bAusgeschalten := FALSE;
				iState := 0;
			END_IF
																								// Manuell-Modus wird eingeschalten
													
			 IF bStarten THEN																		// Objekt führt Prozessdurch
				 iState := 3;
			 END_IF			
	//____________________________________________________________________________________________
	2: // MANUELL
		// DO
		
		// TRANSITION
	
	//____________________________________________________________________________________________
	3: // LAUFEND
		// DO
			// Auswertung von Limit-Wert
			IF sLimitGrenze.Fx <> 0 THEN
				bLimitx := Auswertung(Soll_Wert := sLimitGrenze.Fx, Ist_Wert := Messung.Fx);
			END_IF
			
			IF sLimitGrenze.Fy <> 0 THEN
				bLimity := Auswertung(Soll_Wert := sLimitGrenze.Fy, Ist_Wert := Messung.Fy);
			END_IF
			
			IF sLimitGrenze.Fz <> 0 THEN
				bLimitz := Auswertung(Soll_Wert := sLimitGrenze.Fz, Ist_Wert := Messung.Fz);
			END_IF
			
			// Auswertung von Erreicht-Wert
			IF sErreichtGrenze.Fx <> 0 THEN
				bErreichtx := Auswertung(Soll_Wert := sErreichtGrenze.Fx, Ist_Wert := Messung.Fx);
			END_IF
			
			IF sErreichtGrenze.Fy <> 0 THEN
				bErreichty := Auswertung(Soll_Wert := sErreichtGrenze.Fy, Ist_Wert := Messung.Fy);
			END_IF
			
			IF sErreichtGrenze.Fz <> 0 THEN
				bErreichtz := Auswertung(Soll_Wert := sErreichtGrenze.Fz, Ist_Wert := Messung.Fz);
			END_IF
			
			IF bLimitx OR bLimity OR bLimitz THEN
				bLimit := TRUE;
			ELSE
				bLimit := FALSE;
			END_IF
			
			IF bErreichtx OR bErreichty OR bErreichtz THEN
				bErreicht := TRUE;
			ELSE
				bErreicht := FALSE;
			END_IF
		
		// TRANSITION
			IF bObjektFertig THEN
				bObjektFertig := FALSE;
				iState := 4;
			END_IF
			
			IF bSkillFertig THEN
				iState := 5;
			END_IF
					
			IF bStoppen THEN
				iState := 6;
			END_IF
	
	//____________________________________________________________________________________________
	4: // ABGESCHLOSSEN_INTERN
		// DO
		
		// TRANSITION
			IF bResettenSkill THEN																	// Objekt resetten		
				iState := 1;
			END_IF
	//____________________________________________________________________________________________
	5: // ABGESCHLOSSEN_EXTERN
		// DO																					
			
			Messung.Fx := 0;
			Messung.Fy := 0;
			Messung.Fz := 0;
			Messung.Tx := 0;
			Messung.Ty := 0;
			Messung.Tz := 0;
		
		// TRANSITION
			IF bResettenSkill THEN																	// Objekt resetten
				iState := 1;
			END_IF
	
	//____________________________________________________________________________________________
	6: // GESTOPPT
		// DO
			
			Messung.Fx := 0;
			Messung.Fy := 0;
			Messung.Fz := 0;
			Messung.Tx := 0;
			Messung.Ty := 0;
			Messung.Tz := 0;
		
		// TRANSITION
			IF bResettenSystem THEN																	// Objekt resetten
				iState := 1;
			END_IF
	
	//____________________________________________________________________________________________
	7: // FEHLER
		// DO
			bError := bFehler;
			
		// TRANSITION
			IF bResettenSystem THEN																	// Objekt resetten
				bFehler	 := FALSE;
				bError := FALSE;
				iState := 1;
			END_IF
	
END_CASE

METHOD Auswertung : BOOL
VAR_INPUT
	Soll_Wert			:LREAL;
	Ist_Wert			:LREAL;
END_VAR
IF ABS(Ist_Wert) >= ABS(Soll_Wert) THEN
	Auswertung := TRUE;
ELSE
	Auswertung := FALSE;
END_IF
END_METHOD

PROPERTY P_Erreicht : BOOL
GET
P_Erreicht := bErreicht;
END_GET
END_PROPERTY

PROPERTY P_ErreichtValue : sKraftVariablen
SET
sErreichtGrenze := P_ErreichtValue;
END_SET
END_PROPERTY

PROPERTY P_Limit : BOOL
GET
P_Limit := bLimit;
END_GET
END_PROPERTY

PROPERTY P_LimitValue : sKraftVariablen
SET
sLimitGrenze := P_LimitValue;
END_SET
END_PROPERTY

PROPERTY P_Messdaten : Kraftvariablen
GET
P_Messdaten := Messung;
END_GET
END_PROPERTY

END_FUNCTION_BLOCK

// ---- POUs/03_Systemmodell/Zustandshandling.TcPOU
PROGRAM Zustandshandling
VAR
	iState			:eSystemState;
	
	bEinschalten	:BOOL;
	bAusschalten	:BOOL;
	bStarten		:BOOL;
	bStoppen		:BOOL;
	bFehler			:BOOL;
	bResetten		:BOOL;
	bAbgeschlossen	:BOOL;
END_VAR

GVL.SystemState := iState;

CASE iState OF
	0:	// AUS
			// DO
			IF GVL.Greifer_State = 1 AND GVL.Robot_State = 1 AND GVL.Sensor_State = 1 THEN
				bEinschalten := TRUE;
			END_IF
			
			// TRANSITION
			IF bEinschalten THEN
				bEinschalten := FALSE;
				iState := 1;
			END_IF
		
			
	1:	// BEREIT
			// DO
			IF GVL.Greifer_State = 3 AND GVL.Robot_State = 3 AND GVL.Sensor_State = 3 THEN
				bStarten := TRUE;
			END_IF
			
			IF GVL.Greifer_State = 0 THEN
				bAusschalten := TRUE;
			END_IF
			
			IF GVL.Error THEN
				bFehler := TRUE;
			END_IF
			
			// TRANSITION
			IF bStarten THEN
				bStarten := FALSE;
				iState := 2;
			END_IF
			
			IF bAusschalten THEN
				bAusschalten := FALSE; 
				iState := 0;
			END_IF
			
			IF bFehler THEN
				bFehler := FALSE;
				iState := 4;
			END_IF
			
	2:	// LAUFEND
			// DO
			IF GVL.SystemCommand = 3 THEN
				bStoppen := TRUE;
			END_IF
			
			IF GVL.Greifer_State = 1 AND GVL.Robot_State = 1 AND GVL.Sensor_State = 1  THEN
				bAbgeschlossen := TRUE;
			END_IF
			
			IF GVL.Error THEN
				bFehler := TRUE;
			END_IF
			
			// TRANSITION
			IF bStoppen THEN
				bStoppen := FALSE;
				iState := 3;
			END_IF
			
			IF bAbgeschlossen THEN
				bAbgeschlossen := FALSE;
				iState := 1;
			END_IF
			
			IF bFehler THEN
				bFehler := FALSE;
				iState := 4;
			END_IF
			
	3:	// GESTOPPT
			// DO
			IF GVL.SystemCommand = 4 THEN
				bResetten := TRUE;
			END_IF
			
			// TRANSITION
			IF bResetten THEN
				bResetten := FALSE;
				iState := 1;
			END_IF
			
	4:	// FEHLER
			// DO
			IF GVL.SystemCommand = 4 THEN
				bResetten := TRUE;
			END_IF
			
			// TRANSITION
			IF bResetten THEN
				bResetten := FALSE;
				iState := 1;
			END_IF
			
END_CASE

END_PROGRAM

// ---- POUs/03_Systemmodell/Systemparameter.TcPOU
PROGRAM Systemparameter
VAR
END_VAR

// Lesen
	// Objektzustände
	GVL.Robot_State 		:= Anlage.UR5.P_State;
	GVL.Greifer_State 		:= Anlage.Gripper.P_State;
	GVL.Sensor_State 		:= Anlage.HEX_E.P_State;

// Zuweisen
	// Eigenschaften	
	Anlage.HEX_E.P_LimitValue 		:= GVL.eKraftLimitValue;
	Anlage.HEX_E.P_ErreichtValue 	:= GVL.eKraftErreichtValue;

END_PROGRAM

// ---- POUs/01_Prozessmodell/01_Skills/02_Skills/00_Referenz/Basis_Skill.TcPOU
FUNCTION_BLOCK Basis_Skill EXTENDS GrundstrukturSkill
VAR_INPUT
END_VAR
VAR_OUTPUT
END_VAR
VAR
END_VAR

// Fehlerüberwachung
IF bFehler THEN
	iState := 3;
END_IF

//_______________________________________________________________
// Reaktion auf Input-Variablen:
	// Starten
	fTrigger(CLK := bExecute);
	fSwitch(Set1 := fTrigger.Q);
	
	IF fSwitch.Q1 AND iSysState = 1 THEN
		bStarten := TRUE;
		fSwitch.RESET := TRUE;
	ELSE
		bStarten := FALSE;
		fSwitch.RESET := FALSE;
	END_IF

	// Stoppen
	IF iSysCommand = 3 THEN
		bStoppen := TRUE;
	ELSE 
		bStoppen := FALSE;
	END_IF

	// Resetten 
	IF iSysCommand = 4 THEN
		bResetten := TRUE;
	ELSE
		bResetten := FALSE;
	END_IF

//_______________________________________________________________
// Zustandsmanagement
CASE iState OF 
0: 	// BEREIT
		// DO
		iSkillCommand := 0;
		bDone := FALSE;
		fSwitch.RESET := FALSE;
		
		IF bStarten THEN
			iSkillCommand := 1;																							// Starten des Objektes 
		END_IF	
		
		IF iObjState = 3 THEN
			fSwitch.RESET := TRUE;	
			bGestartet := TRUE;
		END_IF
			
		// TRANSITION	
		IF bGestartet THEN
			bGestartet := FALSE;
			iState := 1;																							// Objekt wurde gestartet
		END_IF
// _________________________________________________________________________________________________________________________
1: 	// LAUFEND
		// DO
		iSkillCommand := 0;
		bBusy := TRUE;																									// Skill wird ausgeführt
		
		IF bTargetReached OR bLimitReached THEN																			// Prüfen ob Prozessziel erreicht wurde
			iSkillCommand := 2;
		END_IF
		
		IF bStoppen THEN																						// Transition wenn System das Orbjekt stoppt
			bBusy := FALSE;																									// Skill wird nicht mehr ausgeführt
			bGestoppt := TRUE;
		END_IF
		
		IF iObjState = 4 THEN																							// Objekt hat Prozess abgeschlossen
			bBusy := FALSE;																									// Skill wird nicht mehr ausgeführt
			bObjektFertig := TRUE;																							// Objekt ist fertig und wieder bereit
		END_IF
		
		IF bLimitReached AND iObjState = 5 THEN																			// Objekt wurde duch Skill gestoppt - LIMIT
			iSkillCommand := 0;																								// Zurücksetzen von Command
			bLimitReached := FALSE;																							// Zurücksetzen von Information	
			bBusy := FALSE;																									// Skill wird nicht mehr ausgeführt
			bLimitErreicht := TRUE;	
		END_IF
		
		IF bTargetReached AND iObjState = 5 THEN																			// Objekt wurde duch Skill gestoppt - LIMIT
			iSkillCommand := 0;																									// Zurücksetzen von Command
			bTargetReached := FALSE;																							// Zurücksetzen von Information	
			bBusy := FALSE;																										// Skill wird nicht mehr ausgeführt
			bWertErreicht := TRUE;	
		END_IF
			
		// TRANSITION 
		IF bGestoppt THEN																								// Transition zu BEREIT
			bGestoppt := FALSE;																							
			iState := 0;
		END_IF
		
		IF bObjektFertig THEN																							// Transition zu ABGESCHLOSSEN
			bObjektFertig := FALSE;																							// Skill wird nicht mehr ausgeführt
			iState := 2;																									// Objekt ist fertig und wieder bereit
		END_IF
		
		IF bLimitErreicht THEN																							// Transition zu LIMIT
			bLimitErreicht := FALSE;
			iState := 4;
		END_IF
		
		IF bWertErreicht THEN																							// Transition zu ERREICHT																						// Skill wird nicht mehr ausgeführt
			bWertErreicht := FALSE;
			iState := 5;
		END_IF
			
// _________________________________________________________________________________________________________________________			
2: 	// ABGESCHLOSSEN
		// DO
		iSkillCommand := 3;																								// Objekt resetten
		bDone := TRUE;																									// Skill wurde erfolgreich ausgeführt
																													
		
		IF iObjState = 1 THEN																							// Objekt wurde geresettet
			iSkillCommand := 0;																								// Zurücksetzen von Command
			bDone := FALSE;																									// Zurücksetzen von Skill
			bSkillFertig := TRUE;									
		END_IF
			
		//  TRANSITION
		IF bSkillFertig THEN
			bSkillFertig := FALSE;																																											// Resetten von Objekt
			iState := 0;
		END_IF
		
// _________________________________________________________________________________________________________________________
3: 	// FEHLER
		// DO 	
		iSkillCommand := 0;
		
		bDone := FALSE;
		bBusy := FALSE;
		
		// TRANSITION
		IF bResetten THEN
			iState := 0;
		END_IF
		
// _________________________________________________________________________________________________________________________			
4: 	// LIMIT
		// DO 
		bLimit := TRUE;																									// Limit wurde erreicht
		
		iSkillCommand := 3;																								// Objekt resetten
		
		IF iObjState = 1 THEN																							// Objekt wurde geresettet
			iSkillCommand := 0;																								// Zurücksetzen von Command
			bDone := FALSE;																									// Zurücksetzen von Skill
			bResetten := TRUE;								
		END_IF
	
		// TRANSITION
		IF bResetten THEN
			bResetten := FALSE;
			bLimit := FALSE;																							// Zurücksetzen von Output-Variable
			iState := 0;
		END_IF
			
// _________________________________________________________________________________________________________________________
5: 	// ERREICHT		
		// DO 
		bDone := TRUE;																									// Skill wurde erfolgreich ausgeführt
		
		iSkillCommand := 3;																								// Objekt resetten
		
		IF iObjState = 1 THEN																							// Objekt wurde geresettet
			iSkillCommand := 0;																								// Zurücksetzen von Command
			bDone := FALSE;																									// Zurücksetzen von Skill
			bSkillFertig := TRUE;									
		END_IF
		
		// TRANSITION
		IF bSkillFertig THEN
			bSkillFertig := FALSE;
			iState := 0;
		END_IF
		
END_CASE

END_FUNCTION_BLOCK

// ---- POUs/01_Prozessmodell/01_Skills/02_Skills/02_Greifer/Skill_Greifer_Oeffnen.TcPOU
FUNCTION_BLOCK Skill_Greifer_Oeffnen EXTENDS GrundstrukturSkill
VAR_INPUT
END_VAR
VAR_OUTPUT
END_VAR
VAR
END_VAR

// Fehlerüberwachung
IF bFehler THEN
	iState := 3;
END_IF

//_______________________________________________________________
// Reaktion auf Input-Variablen:
	// Starten
	fTrigger(CLK := bExecute);
	fSwitch(Set1 := fTrigger.Q);
	
	IF fSwitch.Q1 AND iSysState = 1 THEN
		bStarten := TRUE;
	ELSE
		bStarten := FALSE;
	END_IF

	// Stoppen
	IF iSysCommand = 3 AND iSysState = 2 THEN
		bStoppen := TRUE;
	ELSE 
		bStoppen := FALSE;
	END_IF

	// Resetten 
	IF iSysCommand = 4 THEN
		bResetten := TRUE;
	ELSE
		bResetten := FALSE;
	END_IF

//_______________________________________________________________
// Zustandsmanagement
CASE iState OF 
0: 	// BEREIT
		// DO
		iSkillCommand := 0;
		bDone := FALSE;
		fSwitch.RESET := FALSE;
		
		IF bStarten THEN
			iSkillCommand := 1;																							// Starten des Objektes 
		END_IF	
		
		IF iObjState = 3 THEN
			fSwitch.RESET := TRUE;	
			bGestartet := TRUE;
		END_IF
			
		// TRANSITION	
		IF bGestartet THEN
			bGestartet := FALSE;
			iState := 1;																							// Objekt wurde gestartet
		END_IF
// _________________________________________________________________________________________________________________________
1: 	// LAUFEND
		// DO
		iSkillCommand := 0;
		bBusy := TRUE;																									// Skill wird ausgeführt
		
		IF bTargetReached OR bLimitReached THEN																			// Prüfen ob Prozessziel erreicht wurde
			iSkillCommand := 2;
		END_IF
		
		IF bStoppen THEN																						// Transition wenn System das Orbjekt stoppt
			bBusy := FALSE;																									// Skill wird nicht mehr ausgeführt
			bGestoppt := TRUE;
		END_IF
		
		IF iObjState = 4 THEN																							// Objekt hat Prozess abgeschlossen
			bBusy := FALSE;																									// Skill wird nicht mehr ausgeführt
			bObjektFertig := TRUE;																							// Objekt ist fertig und wieder bereit
		END_IF
		
		IF bLimitReached AND iObjState = 5 THEN																			// Objekt wurde duch Skill gestoppt - LIMIT
			iSkillCommand := 0;																								// Zurücksetzen von Command
			bLimitReached := FALSE;																							// Zurücksetzen von Information	
			bBusy := FALSE;																									// Skill wird nicht mehr ausgeführt
			bLimitErreicht := TRUE;	
		END_IF
		
		IF bTargetReached AND iObjState = 5 THEN																			// Objekt wurde duch Skill gestoppt - LIMIT
			iSkillCommand := 0;																									// Zurücksetzen von Command
			bTargetReached := FALSE;																							// Zurücksetzen von Information	
			bBusy := FALSE;																										// Skill wird nicht mehr ausgeführt
			bWertErreicht := TRUE;	
		END_IF
			
		// TRANSITION 
		IF bGestoppt THEN																								// Transition zu BEREIT
			bGestoppt := FALSE;																							
			iState := 0;
		END_IF
		
		IF bObjektFertig THEN																							// Transition zu ABGESCHLOSSEN
			bObjektFertig := FALSE;																							// Skill wird nicht mehr ausgeführt
			iState := 2;																									// Objekt ist fertig und wieder bereit
		END_IF
		
		IF bLimitErreicht THEN																							// Transition zu LIMIT
			bLimitErreicht := FALSE;
			iState := 4;
		END_IF
		
		IF bWertErreicht THEN																							// Transition zu ERREICHT																						// Skill wird nicht mehr ausgeführt
			bWertErreicht := FALSE;
			iState := 5;
		END_IF
			
// _________________________________________________________________________________________________________________________			
2: 	// ABGESCHLOSSEN
		// DO
		bDone := TRUE;																									// Skill wurde erfolgreich ausgeführt
			
		iSkillCommand := 3;																								// Objekt resetten
		
		IF iObjState = 1 THEN																							// Objekt wurde geresettet
			iSkillCommand := 0;																								// Zurücksetzen von Command
			bDone := FALSE;																									// Zurücksetzen von Skill
			bSkillFertig := TRUE;									
		END_IF
			
		//  TRANSITION
		IF bSkillFertig THEN
			bSkillFertig := FALSE;																																											// Resetten von Objekt
			iState := 0;
		END_IF
		
// _________________________________________________________________________________________________________________________
3: 	// FEHLER
		// DO 	
		iSkillCommand := 0;
		
		bDone := FALSE;
		bBusy := FALSE;
		
		// TRANSITION
		IF bResetten THEN
			iState := 0;
		END_IF
		
// _________________________________________________________________________________________________________________________			
4: 	// LIMIT
		// DO 
		iSkillCommand := 0;
		bLimit := TRUE;																									// Limit wurde erreicht
		
		iSkillCommand := 3;																								// Objekt resetten
		
		IF iObjState = 1 THEN																							// Objekt wurde geresettet
			iSkillCommand := 0;																								// Zurücksetzen von Command
			bDone := FALSE;																									// Zurücksetzen von Skill
			bResetten := TRUE;								
		END_IF
	
		// TRANSITION
		IF bResetten THEN
			bResetten := FALSE;
			bLimit := FALSE;																							// Zurücksetzen von Output-Variable
			iSkillCommand := 3;																							// Resetten von Objekt 
			iState := 0;
		END_IF
			
// _________________________________________________________________________________________________________________________
5: 	// ERREICHT		
		// DO 
		iSkillCommand := 0;
		bDone := TRUE;																									// Skill wurde erfolgreich ausgeführt
		
		iSkillCommand := 3;																								// Objekt resetten
		
		IF iObjState = 1 THEN																							// Objekt wurde geresettet
			iSkillCommand := 0;																								// Zurücksetzen von Command
			bDone := FALSE;																									// Zurücksetzen von Skill
			bSkillFertig := TRUE;									
		END_IF
		
		// TRANSITION
		IF bSkillFertig THEN
			bSkillFertig := FALSE;
			iState := 0;
		END_IF
		
END_CASE

END_FUNCTION_BLOCK

// ---- POUs/01_Prozessmodell/01_Skills/02_Skills/02_Greifer/Skill_Greifer_Pos_Anfahren.TcPOU
FUNCTION_BLOCK Skill_Greifer_Pos_Anfahren EXTENDS GrundstrukturSkill
VAR_INPUT
	sProzessvariablen			:sSmartGreiferProzessVariablen;
END_VAR
VAR_OUTPUT
	sObjektvariablen			:sSmartGreiferProzessVariablen;
END_VAR
VAR
END_VAR

// Fehlerüberwachung
IF bFehler THEN
	iState := 3;
END_IF

//_______________________________________________________________
// Reaktion auf Input-Variablen:
	// Starten
	fTrigger(CLK := bExecute);
	fSwitch(Set1 := fTrigger.Q);
	
	IF fSwitch.Q1 AND iSysState = 1 THEN
		bStarten := TRUE;
	ELSE
		bStarten := FALSE;
	END_IF

	// Stoppen
	IF iSysCommand = 3 AND iSysState = 2 THEN
		bStoppen := TRUE;
	ELSE 
		bStoppen := FALSE;
	END_IF

	// Resetten 
	IF iSysCommand = 4 THEN
		bResetten := TRUE;
	ELSE
		bResetten := FALSE;
	END_IF

//_______________________________________________________________
// Zustandsmanagement
CASE iState OF 
0: 	// BEREIT
		// DO
		iSkillCommand := 0;
		bDone := FALSE;
		fSwitch.RESET := FALSE;
		
		IF bStarten THEN
			sObjektvariablen := sProzessvariablen;
			iSkillCommand := 1;																							// Starten des Objektes 
		END_IF	
		
		IF iObjState = 3 THEN
			fSwitch.RESET := TRUE;	
			bGestartet := TRUE;
		END_IF
			
		// TRANSITION	
		IF bGestartet THEN
			bGestartet := FALSE;
			iState := 1;																							// Objekt wurde gestartet
		END_IF
// _________________________________________________________________________________________________________________________
1: 	// LAUFEND
		// DO
		iSkillCommand := 0;
		bBusy := TRUE;																									// Skill wird ausgeführt
		
		IF bTargetReached OR bLimitReached THEN																			// Prüfen ob Prozessziel erreicht wurde
			iSkillCommand := 2;
		END_IF
		
		IF bStoppen THEN																						// Transition wenn System das Orbjekt stoppt
			bBusy := FALSE;																									// Skill wird nicht mehr ausgeführt
			bGestoppt := TRUE;
		END_IF
		
		IF iObjState = 4 THEN																							// Objekt hat Prozess abgeschlossen
			bBusy := FALSE;																									// Skill wird nicht mehr ausgeführt
			bObjektFertig := TRUE;																							// Objekt ist fertig und wieder bereit
		END_IF
			
		// TRANSITION 
		IF bGestoppt THEN																								// Transition zu BEREIT
			bGestoppt := FALSE;																							
			iState := 0;
		END_IF
		
		IF bObjektFertig THEN																							// Transition zu ABGESCHLOSSEN
			bObjektFertig := FALSE;																							// Skill wird nicht mehr ausgeführt
			iState := 2;																									// Objekt ist fertig und wieder bereit
		END_IF
			
// _________________________________________________________________________________________________________________________			
2: 	// ABGESCHLOSSEN
		// DO
		bDone := TRUE;																									// Skill wurde erfolgreich ausgeführt
			
		iSkillCommand := 3;																								// Objekt resetten
		
		IF iObjState = 1 THEN																							// Objekt wurde geresettet
			iSkillCommand := 0;																								// Zurücksetzen von Command
			bDone := FALSE;																									// Zurücksetzen von Skill
			bSkillFertig := TRUE;									
		END_IF
			
		//  TRANSITION
		IF bSkillFertig THEN
			bSkillFertig := FALSE;																																											// Resetten von Objekt
			iState := 0;
		END_IF
		
// _________________________________________________________________________________________________________________________
3: 	// FEHLER
		// DO 	
		iSkillCommand := 0;
		
		bDone := FALSE;
		bBusy := FALSE;
		
		// TRANSITION
		IF bResetten THEN
			iState := 0;
		END_IF
		
END_CASE

END_FUNCTION_BLOCK

// ---- POUs/01_Prozessmodell/01_Skills/02_Skills/02_Greifer/Skill_Greifer_Schliessen.TcPOU
FUNCTION_BLOCK Skill_Greifer_Schliessen EXTENDS GrundstrukturSkill
VAR_INPUT
END_VAR
VAR_OUTPUT
END_VAR
VAR
END_VAR

// Fehlerüberwachung
IF bFehler THEN
	iState := 3;
END_IF

//_______________________________________________________________
// Reaktion auf Input-Variablen:
	// Starten
	fTrigger(CLK := bExecute);
	fSwitch(Set1 := fTrigger.Q);
	
	IF fSwitch.Q1 AND iSysState = 1 THEN
		bStarten := TRUE;
	ELSE
		bStarten := FALSE;
	END_IF

	// Stoppen
	IF iSysCommand = 3 AND iSysState = 2 THEN
		bStoppen := TRUE;
	ELSE 
		bStoppen := FALSE;
	END_IF

	// Resetten 
	IF iSysCommand = 4 THEN
		bResetten := TRUE;
	ELSE
		bResetten := FALSE;
	END_IF

//_______________________________________________________________
// Zustandsmanagement
CASE iState OF 
0: 	// BEREIT
		// DO
		iSkillCommand := 0;
		bDone := FALSE;
		fSwitch.RESET := FALSE;
		
		IF bStarten THEN
			iSkillCommand := 1;																							// Starten des Objektes 
		END_IF	
		
		IF iObjState = 3 THEN
			fSwitch.RESET := TRUE;	
			bGestartet := TRUE;
		END_IF
			
		// TRANSITION	
		IF bGestartet THEN
			bGestartet := FALSE;
			iState := 1;																							// Objekt wurde gestartet
		END_IF
// _________________________________________________________________________________________________________________________
1: 	// LAUFEND
		// DO
		iSkillCommand := 0;
		bBusy := TRUE;																									// Skill wird ausgeführt
		
		IF bTargetReached OR bLimitReached THEN																			// Prüfen ob Prozessziel erreicht wurde
			iSkillCommand := 2;
		END_IF
		
		IF bStoppen THEN																						// Transition wenn System das Orbjekt stoppt
			bBusy := FALSE;																									// Skill wird nicht mehr ausgeführt
			bGestoppt := TRUE;
		END_IF
		
		IF iObjState = 4 THEN																							// Objekt hat Prozess abgeschlossen
			bBusy := FALSE;																									// Skill wird nicht mehr ausgeführt
			bObjektFertig := TRUE;																							// Objekt ist fertig und wieder bereit
		END_IF
		
		IF bLimitReached AND iObjState = 5 THEN																			// Objekt wurde duch Skill gestoppt - LIMIT
			iSkillCommand := 0;																								// Zurücksetzen von Command
			bLimitReached := FALSE;																							// Zurücksetzen von Information	
			bBusy := FALSE;																									// Skill wird nicht mehr ausgeführt
			bLimitErreicht := TRUE;	
		END_IF
		
		IF bTargetReached AND iObjState = 5 THEN																			// Objekt wurde duch Skill gestoppt - LIMIT
			iSkillCommand := 0;																									// Zurücksetzen von Command
			bTargetReached := FALSE;																							// Zurücksetzen von Information	
			bBusy := FALSE;																										// Skill wird nicht mehr ausgeführt
			bWertErreicht := TRUE;	
		END_IF
			
		// TRANSITION 
		IF bGestoppt THEN																								// Transition zu BEREIT
			bGestoppt := FALSE;																							
			iState := 0;
		END_IF
		
		IF bObjektFertig THEN																							// Transition zu ABGESCHLOSSEN
			bObjektFertig := FALSE;																							// Skill wird nicht mehr ausgeführt
			iState := 2;																									// Objekt ist fertig und wieder bereit
		END_IF
		
		IF bLimitErreicht THEN																							// Transition zu LIMIT
			bLimitErreicht := FALSE;
			iState := 4;
		END_IF
		
		IF bWertErreicht THEN																							// Transition zu ERREICHT																						// Skill wird nicht mehr ausgeführt
			bWertErreicht := FALSE;
			iState := 5;
		END_IF
			
// _________________________________________________________________________________________________________________________			
2: 	// ABGESCHLOSSEN
		// DO
		bDone := TRUE;																									// Skill wurde erfolgreich ausgeführt
			
		iSkillCommand := 3;																								// Objekt resetten
		
